// TIA Portal V17 export
// export: Created 2023-04-06T09:22:57.7461834Z, ExportSetting WithDefaults, DisplayName Totally Integrated Automation Portal, DisplayVersion V17 Update 4, DisplayName TIA Portal Openness, DisplayVersion V17 Update 4, DisplayName TIA Portal Version Control Interface, DisplayVersion V17, DisplayName STEP 7 Professional, DisplayVersion V17 Update 4, DisplayName STEP 7 Safety, DisplayVersion V17, DisplayName WinCC Professional, DisplayVersion V17 Update 4
FUNCTION "BMS 1 (S)" : Void   // FC25, LAD
TITLE = ModBus TCP for CATL Battery
{ S7_Optimized_Access := 'TRUE' }
VERSION : 0.1
// stored: AutoNumber false, IsIECCheckEnabled false, SetENOAutomatically false, UDAEnableTagReadback false
   VAR_TEMP
      xSpare : Bool;
      BBwAlm1 : Word;
      BBwWarn1 : Word;
      BR01wAlm1 : Word;
      BR01wAlm2 : Word;
      BR01wAlm3 : Word;
      BR01wWarn1 : Word;
      BR02wAlm1 : Word;
      BR02wAlm2 : Word;
      BR02wAlm3 : Word;
      BR02wWarn1 : Word;
      BR03wAlm1 : Word;
      BR03wAlm2 : Word;
      BR03wAlm3 : Word;
      BR03wWarn1 : Word;
      BR04wAlm1 : Word;
      BR04wAlm2 : Word;
      BR04wAlm3 : Word;
      BR04wWarn1 : Word;
      BR05wAlm1 : Word;
      BR05wAlm2 : Word;
      BR05wAlm3 : Word;
      BR05wWarn1 : Word;
      BR06wAlm1 : Word;
      BR06wAlm2 : Word;
      BR06wAlm3 : Word;
      BR06wWarn1 : Word;
      BR07wAlm1 : Word;
      BR07wAlm2 : Word;
      BR07wAlm3 : Word;
      BR07wWarn1 : Word;
      BR08wAlm1 : Word;
      BR08wAlm2 : Word;
      BR08wAlm3 : Word;
      BR08wWarn1 : Word;
      BR09wAlm1 : Word;
      BR09wAlm2 : Word;
      BR09wAlm3 : Word;
      BR09wWarn1 : Word;
      BR10wAlm1 : Word;
      BR10wAlm2 : Word;
      BR10wAlm3 : Word;
      BR10wWarn1 : Word;
      BR11wAlm1 : Word;
      BR11wAlm2 : Word;
      BR11wAlm3 : Word;
      BR11wWarn1 : Word;
      BR12wAlm1 : Word;
      BR12wAlm2 : Word;
      BR12wAlm3 : Word;
      BR12wWarn1 : Word;
   END_VAR
   VAR_TEMP   // added for the SCL form of the ladder/FBD networks
      _w1 : Bool;
   END_VAR
BEGIN

REGION Network 1: Function Modbus Client
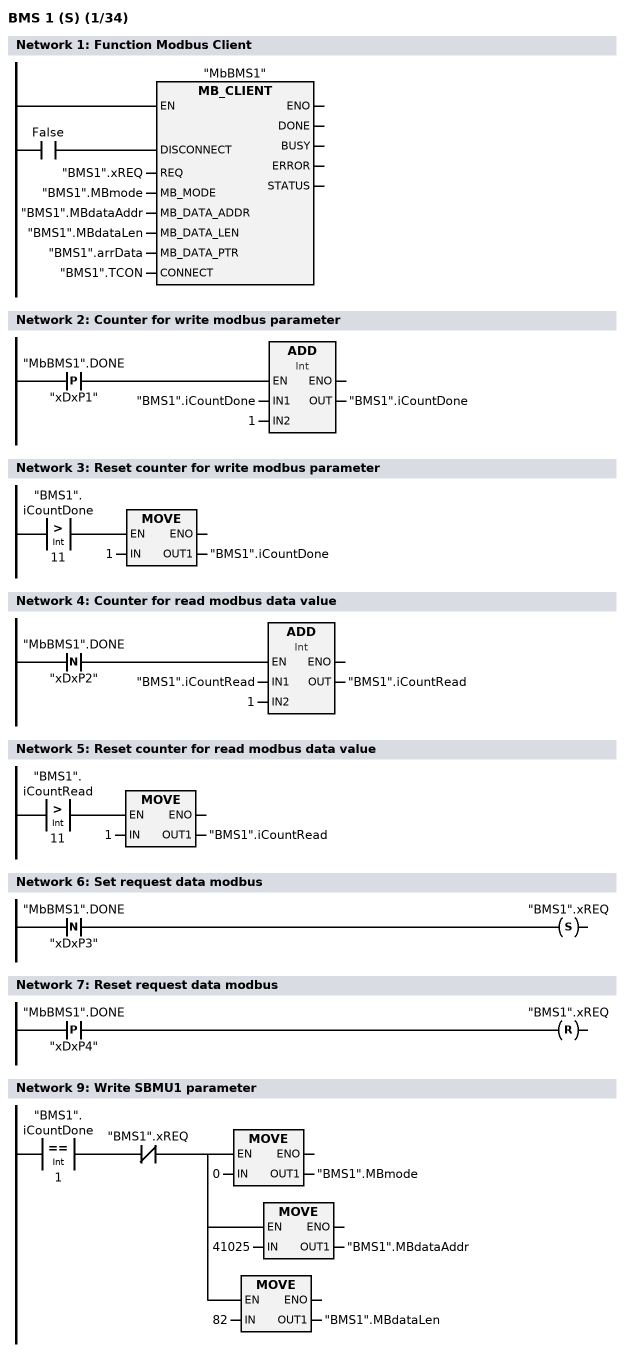
   RUNG wire#powerrail
      "MbBMS1".MB_CLIENT(DISCONNECT := wire#w1, REQ := "BMS1".xREQ, MB_MODE := "BMS1".MBmode, MB_DATA_ADDR := "BMS1".MBdataAddr, MB_DATA_LEN := "BMS1".MBdataLen, MB_DATA_PTR := "BMS1".arrData, CONNECT := "BMS1".TCON, DONE =>, BUSY =>, ERROR =>, STATUS =>)
   END_RUNG
   RUNG wire#powerrail
      Contact( False )
   END_RUNG wire#w1
   // the same network as SCL:
   "MbBMS1"(DISCONNECT := False,   // MB_CLIENT
            REQ := "BMS1".xREQ,
            MB_MODE := "BMS1".MBmode,
            MB_DATA_ADDR := "BMS1".MBdataAddr,
            MB_DATA_LEN := "BMS1".MBdataLen,
            MB_DATA_PTR := "BMS1".arrData,
            CONNECT := "BMS1".TCON);
END_REGION

REGION Network 2: Counter for write modbus parameter
   RUNG wire#powerrail
      P_Contact(operand := "MbBMS1".DONE, bit := "xDxP1")
      { S7_Templates := "SrcType := Int" } Add(in1 := "BMS1".iCountDone, in2 := 1, out => "BMS1".iCountDone)
   END_RUNG
   // the same network as SCL:
   #_w1 := "MbBMS1".DONE AND NOT "xDxP1";   // rising edge of "MbBMS1".DONE
   "xDxP1" := "MbBMS1".DONE;
   IF #_w1 THEN "BMS1".iCountDone := "BMS1".iCountDone + 1; END_IF;
END_REGION

REGION Network 3: Reset counter for write modbus parameter
   RUNG wire#powerrail
      { S7_Templates := "SrcType := Int" } GT_Contact(in1 := "BMS1".iCountDone, in2 := 11)
      Move(in := 1, out1 => "BMS1".iCountDone)
   END_RUNG
   // the same network as SCL:
   IF "BMS1".iCountDone > 11 THEN "BMS1".iCountDone := 1; END_IF;
END_REGION

REGION Network 4: Counter for read modbus data value
   RUNG wire#powerrail
      N_Contact(operand := "MbBMS1".DONE, bit := "xDxP2")
      { S7_Templates := "SrcType := Int" } Add(in1 := "BMS1".iCountRead, in2 := 1, out => "BMS1".iCountRead)
   END_RUNG
   // the same network as SCL:
   #_w1 := NOT "MbBMS1".DONE AND "xDxP2";   // falling edge of "MbBMS1".DONE
   "xDxP2" := "MbBMS1".DONE;
   IF #_w1 THEN "BMS1".iCountRead := "BMS1".iCountRead + 1; END_IF;
END_REGION

REGION Network 5: Reset counter for read modbus data value
   RUNG wire#powerrail
      { S7_Templates := "SrcType := Int" } GT_Contact(in1 := "BMS1".iCountRead, in2 := 11)
      Move(in := 1, out1 => "BMS1".iCountRead)
   END_RUNG
   // the same network as SCL:
   IF "BMS1".iCountRead > 11 THEN "BMS1".iCountRead := 1; END_IF;
END_REGION

REGION Network 6: Set request data modbus
   RUNG wire#powerrail
      N_Contact(operand := "MbBMS1".DONE, bit := "xDxP3")
      S_Coil( "BMS1".xREQ )
   END_RUNG
   // the same network as SCL:
   #_w1 := NOT "MbBMS1".DONE AND "xDxP3";   // falling edge of "MbBMS1".DONE
   "xDxP3" := "MbBMS1".DONE;
   IF #_w1 THEN "BMS1".xREQ := TRUE; END_IF;
END_REGION

REGION Network 7: Reset request data modbus
   RUNG wire#powerrail
      P_Contact(operand := "MbBMS1".DONE, bit := "xDxP4")
      R_Coil( "BMS1".xREQ )
   END_RUNG
   // the same network as SCL:
   #_w1 := "MbBMS1".DONE AND NOT "xDxP4";   // rising edge of "MbBMS1".DONE
   "xDxP4" := "MbBMS1".DONE;
   IF #_w1 THEN "BMS1".xREQ := FALSE; END_IF;
END_REGION

REGION Network 9: Write SBMU1 parameter
   RUNG wire#powerrail
      { S7_Templates := "SrcType := Int" } EQ_Contact(in1 := "BMS1".iCountDone, in2 := 1)
      I_Contact( "BMS1".xREQ )
      wire#w1
      Move(in := 0, out1 => "BMS1".MBmode)
   END_RUNG
   RUNG wire#w1
      Move(in := 41025, out1 => "BMS1".MBdataAddr)
   END_RUNG
   RUNG wire#w1
      Move(in := 82, out1 => "BMS1".MBdataLen)
   END_RUNG
   // the same network as SCL:
   IF ("BMS1".iCountDone = 1) AND NOT "BMS1".xREQ THEN
       "BMS1".MBmode := 0;
       "BMS1".MBdataAddr := 41025;
       "BMS1".MBdataLen := 82;
   END_IF;
END_REGION

REGION Network 10: Read SBMU1 data value
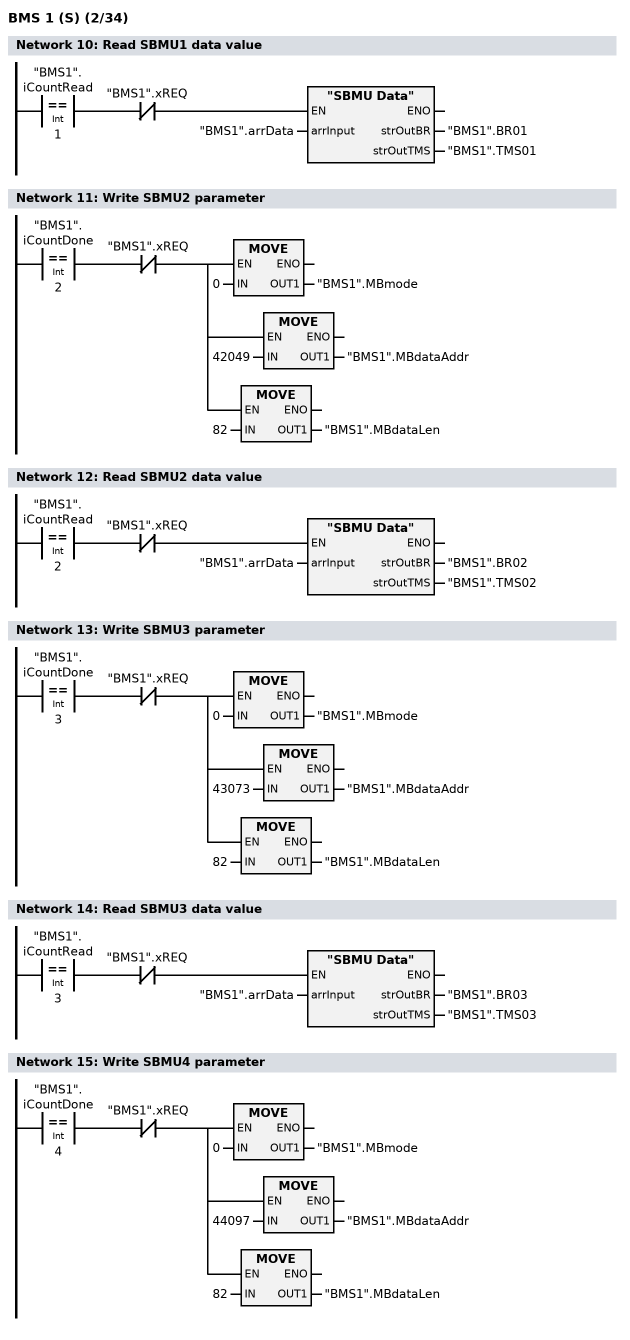
   RUNG wire#powerrail
      { S7_Templates := "SrcType := Int" } EQ_Contact(in1 := "BMS1".iCountRead, in2 := 1)
      I_Contact( "BMS1".xREQ )
      "SBMU Data"(arrInput := "BMS1".arrData, strOutBR => "BMS1".BR01, strOutTMS => "BMS1".TMS01)
   END_RUNG
   // the same network as SCL:
   IF ("BMS1".iCountRead = 1) AND NOT "BMS1".xREQ THEN
       "SBMU Data"(arrInput := "BMS1".arrData, strOutBR => "BMS1".BR01, strOutTMS => "BMS1".TMS01);
   END_IF;
END_REGION

REGION Network 11: Write SBMU2 parameter
   RUNG wire#powerrail
      { S7_Templates := "SrcType := Int" } EQ_Contact(in1 := "BMS1".iCountDone, in2 := 2)
      I_Contact( "BMS1".xREQ )
      wire#w1
      Move(in := 0, out1 => "BMS1".MBmode)
   END_RUNG
   RUNG wire#w1
      Move(in := 42049, out1 => "BMS1".MBdataAddr)
   END_RUNG
   RUNG wire#w1
      Move(in := 82, out1 => "BMS1".MBdataLen)
   END_RUNG
   // the same network as SCL:
   IF ("BMS1".iCountDone = 2) AND NOT "BMS1".xREQ THEN
       "BMS1".MBmode := 0;
       "BMS1".MBdataAddr := 42049;
       "BMS1".MBdataLen := 82;
   END_IF;
END_REGION

REGION Network 12: Read SBMU2 data value
   RUNG wire#powerrail
      { S7_Templates := "SrcType := Int" } EQ_Contact(in1 := "BMS1".iCountRead, in2 := 2)
      I_Contact( "BMS1".xREQ )
      "SBMU Data"(arrInput := "BMS1".arrData, strOutBR => "BMS1".BR02, strOutTMS => "BMS1".TMS02)
   END_RUNG
   // the same network as SCL:
   IF ("BMS1".iCountRead = 2) AND NOT "BMS1".xREQ THEN
       "SBMU Data"(arrInput := "BMS1".arrData, strOutBR => "BMS1".BR02, strOutTMS => "BMS1".TMS02);
   END_IF;
END_REGION

REGION Network 13: Write SBMU3 parameter
   RUNG wire#powerrail
      { S7_Templates := "SrcType := Int" } EQ_Contact(in1 := "BMS1".iCountDone, in2 := 3)
      I_Contact( "BMS1".xREQ )
      wire#w1
      Move(in := 0, out1 => "BMS1".MBmode)
   END_RUNG
   RUNG wire#w1
      Move(in := 43073, out1 => "BMS1".MBdataAddr)
   END_RUNG
   RUNG wire#w1
      Move(in := 82, out1 => "BMS1".MBdataLen)
   END_RUNG
   // the same network as SCL:
   IF ("BMS1".iCountDone = 3) AND NOT "BMS1".xREQ THEN
       "BMS1".MBmode := 0;
       "BMS1".MBdataAddr := 43073;
       "BMS1".MBdataLen := 82;
   END_IF;
END_REGION

REGION Network 14: Read SBMU3 data value
   RUNG wire#powerrail
      { S7_Templates := "SrcType := Int" } EQ_Contact(in1 := "BMS1".iCountRead, in2 := 3)
      I_Contact( "BMS1".xREQ )
      "SBMU Data"(arrInput := "BMS1".arrData, strOutBR => "BMS1".BR03, strOutTMS => "BMS1".TMS03)
   END_RUNG
   // the same network as SCL:
   IF ("BMS1".iCountRead = 3) AND NOT "BMS1".xREQ THEN
       "SBMU Data"(arrInput := "BMS1".arrData, strOutBR => "BMS1".BR03, strOutTMS => "BMS1".TMS03);
   END_IF;
END_REGION

REGION Network 15: Write SBMU4 parameter
   RUNG wire#powerrail
      { S7_Templates := "SrcType := Int" } EQ_Contact(in1 := "BMS1".iCountDone, in2 := 4)
      I_Contact( "BMS1".xREQ )
      wire#w1
      Move(in := 0, out1 => "BMS1".MBmode)
   END_RUNG
   RUNG wire#w1
      Move(in := 44097, out1 => "BMS1".MBdataAddr)
   END_RUNG
   RUNG wire#w1
      Move(in := 82, out1 => "BMS1".MBdataLen)
   END_RUNG
   // the same network as SCL:
   IF ("BMS1".iCountDone = 4) AND NOT "BMS1".xREQ THEN
       "BMS1".MBmode := 0;
       "BMS1".MBdataAddr := 44097;
       "BMS1".MBdataLen := 82;
   END_IF;
END_REGION

REGION Network 16: Read SBMU4 data value
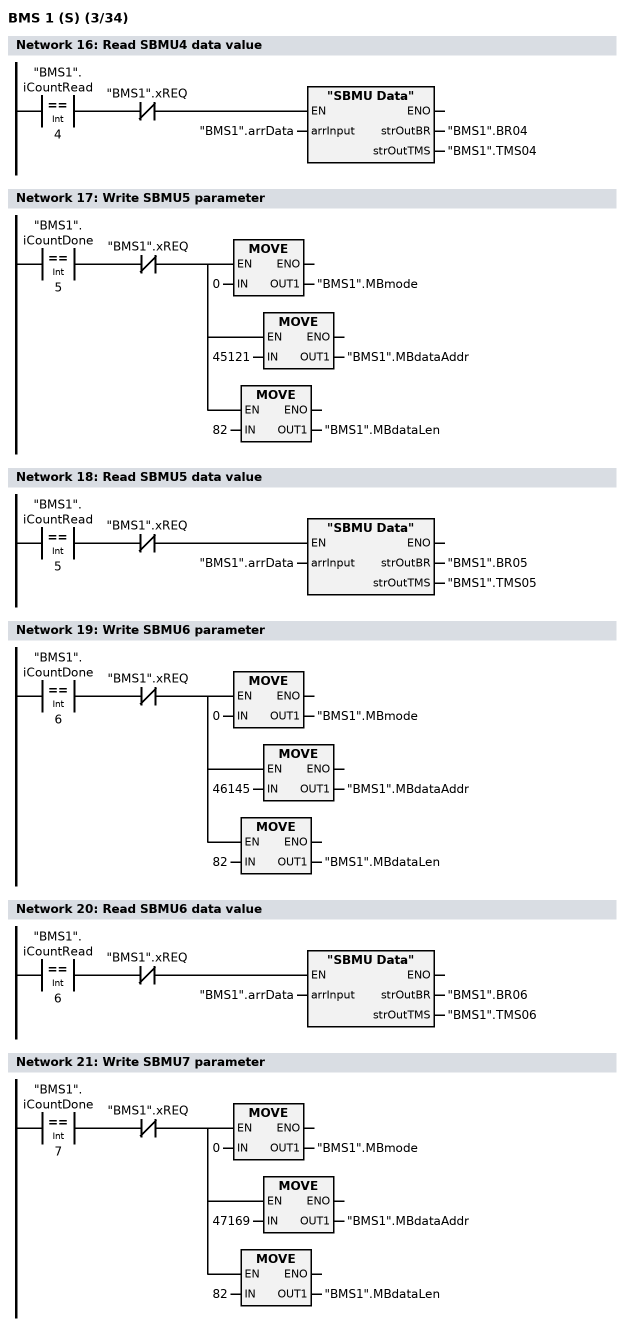
   RUNG wire#powerrail
      { S7_Templates := "SrcType := Int" } EQ_Contact(in1 := "BMS1".iCountRead, in2 := 4)
      I_Contact( "BMS1".xREQ )
      "SBMU Data"(arrInput := "BMS1".arrData, strOutBR => "BMS1".BR04, strOutTMS => "BMS1".TMS04)
   END_RUNG
   // the same network as SCL:
   IF ("BMS1".iCountRead = 4) AND NOT "BMS1".xREQ THEN
       "SBMU Data"(arrInput := "BMS1".arrData, strOutBR => "BMS1".BR04, strOutTMS => "BMS1".TMS04);
   END_IF;
END_REGION

REGION Network 17: Write SBMU5 parameter
   RUNG wire#powerrail
      { S7_Templates := "SrcType := Int" } EQ_Contact(in1 := "BMS1".iCountDone, in2 := 5)
      I_Contact( "BMS1".xREQ )
      wire#w1
      Move(in := 0, out1 => "BMS1".MBmode)
   END_RUNG
   RUNG wire#w1
      Move(in := 45121, out1 => "BMS1".MBdataAddr)
   END_RUNG
   RUNG wire#w1
      Move(in := 82, out1 => "BMS1".MBdataLen)
   END_RUNG
   // the same network as SCL:
   IF ("BMS1".iCountDone = 5) AND NOT "BMS1".xREQ THEN
       "BMS1".MBmode := 0;
       "BMS1".MBdataAddr := 45121;
       "BMS1".MBdataLen := 82;
   END_IF;
END_REGION

REGION Network 18: Read SBMU5 data value
   RUNG wire#powerrail
      { S7_Templates := "SrcType := Int" } EQ_Contact(in1 := "BMS1".iCountRead, in2 := 5)
      I_Contact( "BMS1".xREQ )
      "SBMU Data"(arrInput := "BMS1".arrData, strOutBR => "BMS1".BR05, strOutTMS => "BMS1".TMS05)
   END_RUNG
   // the same network as SCL:
   IF ("BMS1".iCountRead = 5) AND NOT "BMS1".xREQ THEN
       "SBMU Data"(arrInput := "BMS1".arrData, strOutBR => "BMS1".BR05, strOutTMS => "BMS1".TMS05);
   END_IF;
END_REGION

REGION Network 19: Write SBMU6 parameter
   RUNG wire#powerrail
      { S7_Templates := "SrcType := Int" } EQ_Contact(in1 := "BMS1".iCountDone, in2 := 6)
      I_Contact( "BMS1".xREQ )
      wire#w1
      Move(in := 0, out1 => "BMS1".MBmode)
   END_RUNG
   RUNG wire#w1
      Move(in := 46145, out1 => "BMS1".MBdataAddr)
   END_RUNG
   RUNG wire#w1
      Move(in := 82, out1 => "BMS1".MBdataLen)
   END_RUNG
   // the same network as SCL:
   IF ("BMS1".iCountDone = 6) AND NOT "BMS1".xREQ THEN
       "BMS1".MBmode := 0;
       "BMS1".MBdataAddr := 46145;
       "BMS1".MBdataLen := 82;
   END_IF;
END_REGION

REGION Network 20: Read SBMU6 data value
   RUNG wire#powerrail
      { S7_Templates := "SrcType := Int" } EQ_Contact(in1 := "BMS1".iCountRead, in2 := 6)
      I_Contact( "BMS1".xREQ )
      "SBMU Data"(arrInput := "BMS1".arrData, strOutBR => "BMS1".BR06, strOutTMS => "BMS1".TMS06)
   END_RUNG
   // the same network as SCL:
   IF ("BMS1".iCountRead = 6) AND NOT "BMS1".xREQ THEN
       "SBMU Data"(arrInput := "BMS1".arrData, strOutBR => "BMS1".BR06, strOutTMS => "BMS1".TMS06);
   END_IF;
END_REGION

REGION Network 21: Write SBMU7 parameter
   RUNG wire#powerrail
      { S7_Templates := "SrcType := Int" } EQ_Contact(in1 := "BMS1".iCountDone, in2 := 7)
      I_Contact( "BMS1".xREQ )
      wire#w1
      Move(in := 0, out1 => "BMS1".MBmode)
   END_RUNG
   RUNG wire#w1
      Move(in := 47169, out1 => "BMS1".MBdataAddr)
   END_RUNG
   RUNG wire#w1
      Move(in := 82, out1 => "BMS1".MBdataLen)
   END_RUNG
   // the same network as SCL:
   IF ("BMS1".iCountDone = 7) AND NOT "BMS1".xREQ THEN
       "BMS1".MBmode := 0;
       "BMS1".MBdataAddr := 47169;
       "BMS1".MBdataLen := 82;
   END_IF;
END_REGION

REGION Network 22: Read SBMU7 data value
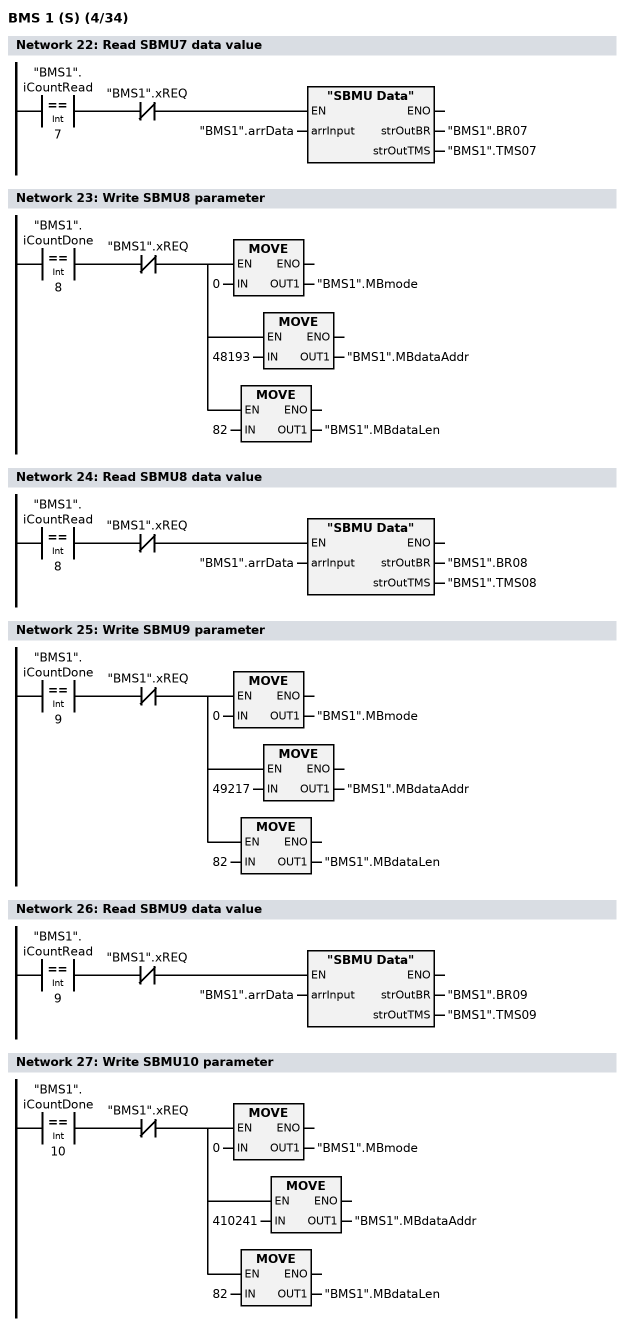
   RUNG wire#powerrail
      { S7_Templates := "SrcType := Int" } EQ_Contact(in1 := "BMS1".iCountRead, in2 := 7)
      I_Contact( "BMS1".xREQ )
      "SBMU Data"(arrInput := "BMS1".arrData, strOutBR => "BMS1".BR07, strOutTMS => "BMS1".TMS07)
   END_RUNG
   // the same network as SCL:
   IF ("BMS1".iCountRead = 7) AND NOT "BMS1".xREQ THEN
       "SBMU Data"(arrInput := "BMS1".arrData, strOutBR => "BMS1".BR07, strOutTMS => "BMS1".TMS07);
   END_IF;
END_REGION

REGION Network 23: Write SBMU8 parameter
   RUNG wire#powerrail
      { S7_Templates := "SrcType := Int" } EQ_Contact(in1 := "BMS1".iCountDone, in2 := 8)
      I_Contact( "BMS1".xREQ )
      wire#w1
      Move(in := 0, out1 => "BMS1".MBmode)
   END_RUNG
   RUNG wire#w1
      Move(in := 48193, out1 => "BMS1".MBdataAddr)
   END_RUNG
   RUNG wire#w1
      Move(in := 82, out1 => "BMS1".MBdataLen)
   END_RUNG
   // the same network as SCL:
   IF ("BMS1".iCountDone = 8) AND NOT "BMS1".xREQ THEN
       "BMS1".MBmode := 0;
       "BMS1".MBdataAddr := 48193;
       "BMS1".MBdataLen := 82;
   END_IF;
END_REGION

REGION Network 24: Read SBMU8 data value
   RUNG wire#powerrail
      { S7_Templates := "SrcType := Int" } EQ_Contact(in1 := "BMS1".iCountRead, in2 := 8)
      I_Contact( "BMS1".xREQ )
      "SBMU Data"(arrInput := "BMS1".arrData, strOutBR => "BMS1".BR08, strOutTMS => "BMS1".TMS08)
   END_RUNG
   // the same network as SCL:
   IF ("BMS1".iCountRead = 8) AND NOT "BMS1".xREQ THEN
       "SBMU Data"(arrInput := "BMS1".arrData, strOutBR => "BMS1".BR08, strOutTMS => "BMS1".TMS08);
   END_IF;
END_REGION

REGION Network 25: Write SBMU9 parameter
   RUNG wire#powerrail
      { S7_Templates := "SrcType := Int" } EQ_Contact(in1 := "BMS1".iCountDone, in2 := 9)
      I_Contact( "BMS1".xREQ )
      wire#w1
      Move(in := 0, out1 => "BMS1".MBmode)
   END_RUNG
   RUNG wire#w1
      Move(in := 49217, out1 => "BMS1".MBdataAddr)
   END_RUNG
   RUNG wire#w1
      Move(in := 82, out1 => "BMS1".MBdataLen)
   END_RUNG
   // the same network as SCL:
   IF ("BMS1".iCountDone = 9) AND NOT "BMS1".xREQ THEN
       "BMS1".MBmode := 0;
       "BMS1".MBdataAddr := 49217;
       "BMS1".MBdataLen := 82;
   END_IF;
END_REGION

REGION Network 26: Read SBMU9 data value
   RUNG wire#powerrail
      { S7_Templates := "SrcType := Int" } EQ_Contact(in1 := "BMS1".iCountRead, in2 := 9)
      I_Contact( "BMS1".xREQ )
      "SBMU Data"(arrInput := "BMS1".arrData, strOutBR => "BMS1".BR09, strOutTMS => "BMS1".TMS09)
   END_RUNG
   // the same network as SCL:
   IF ("BMS1".iCountRead = 9) AND NOT "BMS1".xREQ THEN
       "SBMU Data"(arrInput := "BMS1".arrData, strOutBR => "BMS1".BR09, strOutTMS => "BMS1".TMS09);
   END_IF;
END_REGION

REGION Network 27: Write SBMU10 parameter
   RUNG wire#powerrail
      { S7_Templates := "SrcType := Int" } EQ_Contact(in1 := "BMS1".iCountDone, in2 := 10)
      I_Contact( "BMS1".xREQ )
      wire#w1
      Move(in := 0, out1 => "BMS1".MBmode)
   END_RUNG
   RUNG wire#w1
      Move(in := 410241, out1 => "BMS1".MBdataAddr)
   END_RUNG
   RUNG wire#w1
      Move(in := 82, out1 => "BMS1".MBdataLen)
   END_RUNG
   // the same network as SCL:
   IF ("BMS1".iCountDone = 10) AND NOT "BMS1".xREQ THEN
       "BMS1".MBmode := 0;
       "BMS1".MBdataAddr := 410241;
       "BMS1".MBdataLen := 82;
   END_IF;
END_REGION

REGION Network 28: Read SBMU10 data value
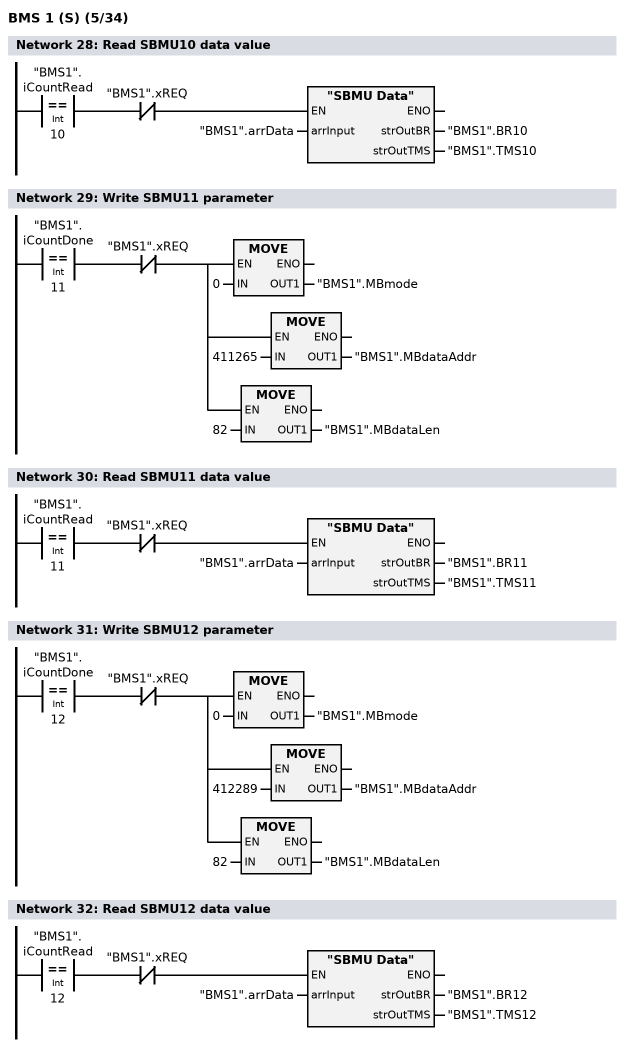
   RUNG wire#powerrail
      { S7_Templates := "SrcType := Int" } EQ_Contact(in1 := "BMS1".iCountRead, in2 := 10)
      I_Contact( "BMS1".xREQ )
      "SBMU Data"(arrInput := "BMS1".arrData, strOutBR => "BMS1".BR10, strOutTMS => "BMS1".TMS10)
   END_RUNG
   // the same network as SCL:
   IF ("BMS1".iCountRead = 10) AND NOT "BMS1".xREQ THEN
       "SBMU Data"(arrInput := "BMS1".arrData, strOutBR => "BMS1".BR10, strOutTMS => "BMS1".TMS10);
   END_IF;
END_REGION

REGION Network 29: Write SBMU11 parameter
   RUNG wire#powerrail
      { S7_Templates := "SrcType := Int" } EQ_Contact(in1 := "BMS1".iCountDone, in2 := 11)
      I_Contact( "BMS1".xREQ )
      wire#w1
      Move(in := 0, out1 => "BMS1".MBmode)
   END_RUNG
   RUNG wire#w1
      Move(in := 411265, out1 => "BMS1".MBdataAddr)
   END_RUNG
   RUNG wire#w1
      Move(in := 82, out1 => "BMS1".MBdataLen)
   END_RUNG
   // the same network as SCL:
   IF ("BMS1".iCountDone = 11) AND NOT "BMS1".xREQ THEN
       "BMS1".MBmode := 0;
       "BMS1".MBdataAddr := 411265;
       "BMS1".MBdataLen := 82;
   END_IF;
END_REGION

REGION Network 30: Read SBMU11 data value
   RUNG wire#powerrail
      { S7_Templates := "SrcType := Int" } EQ_Contact(in1 := "BMS1".iCountRead, in2 := 11)
      I_Contact( "BMS1".xREQ )
      "SBMU Data"(arrInput := "BMS1".arrData, strOutBR => "BMS1".BR11, strOutTMS => "BMS1".TMS11)
   END_RUNG
   // the same network as SCL:
   IF ("BMS1".iCountRead = 11) AND NOT "BMS1".xREQ THEN
       "SBMU Data"(arrInput := "BMS1".arrData, strOutBR => "BMS1".BR11, strOutTMS => "BMS1".TMS11);
   END_IF;
END_REGION

REGION Network 31: Write SBMU12 parameter
   RUNG wire#powerrail
      { S7_Templates := "SrcType := Int" } EQ_Contact(in1 := "BMS1".iCountDone, in2 := 12)
      I_Contact( "BMS1".xREQ )
      wire#w1
      Move(in := 0, out1 => "BMS1".MBmode)
   END_RUNG
   RUNG wire#w1
      Move(in := 412289, out1 => "BMS1".MBdataAddr)
   END_RUNG
   RUNG wire#w1
      Move(in := 82, out1 => "BMS1".MBdataLen)
   END_RUNG
   // the same network as SCL:
   IF ("BMS1".iCountDone = 12) AND NOT "BMS1".xREQ THEN
       "BMS1".MBmode := 0;
       "BMS1".MBdataAddr := 412289;
       "BMS1".MBdataLen := 82;
   END_IF;
END_REGION

REGION Network 32: Read SBMU12 data value
   RUNG wire#powerrail
      { S7_Templates := "SrcType := Int" } EQ_Contact(in1 := "BMS1".iCountRead, in2 := 12)
      I_Contact( "BMS1".xREQ )
      "SBMU Data"(arrInput := "BMS1".arrData, strOutBR => "BMS1".BR12, strOutTMS => "BMS1".TMS12)
   END_RUNG
   // the same network as SCL:
   IF ("BMS1".iCountRead = 12) AND NOT "BMS1".xREQ THEN
       "SBMU Data"(arrInput := "BMS1".arrData, strOutBR => "BMS1".BR12, strOutTMS => "BMS1".TMS12);
   END_IF;
END_REGION

REGION Network 34: Write Command from EMS
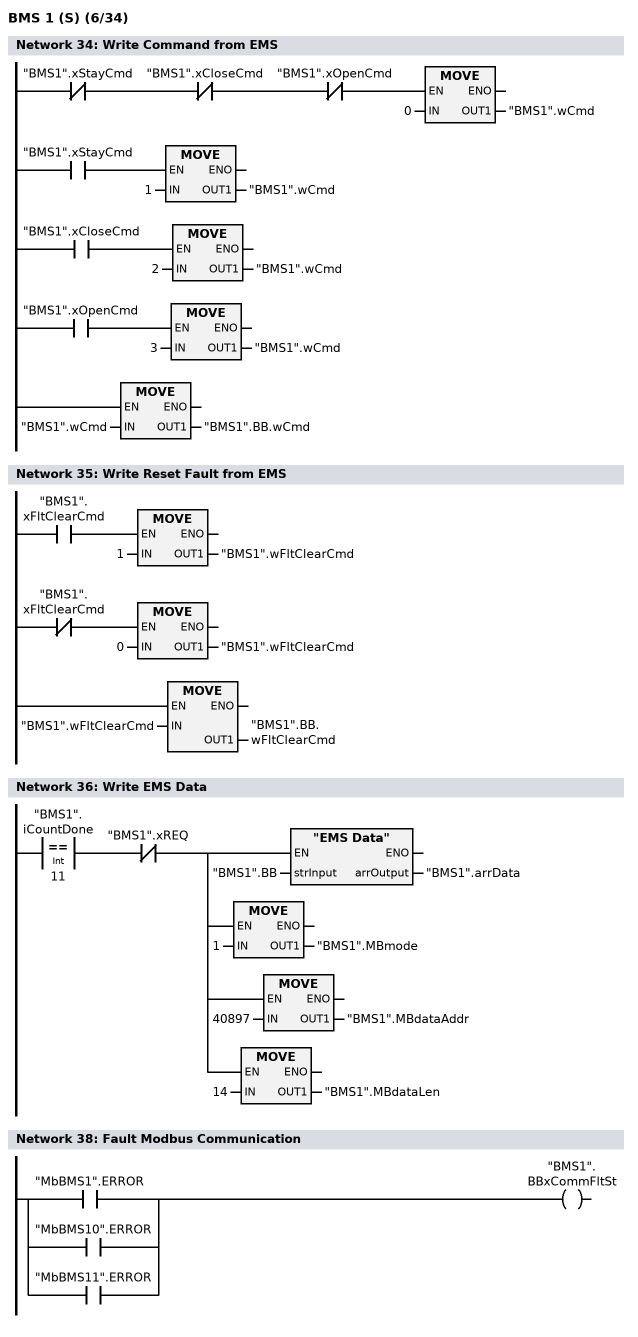
   RUNG wire#powerrail
      I_Contact( "BMS1".xStayCmd )
      I_Contact( "BMS1".xCloseCmd )
      I_Contact( "BMS1".xOpenCmd )
      Move(in := 0, out1 => "BMS1".wCmd)
   END_RUNG
   RUNG wire#powerrail
      Contact( "BMS1".xStayCmd )
      Move(in := 1, out1 => "BMS1".wCmd)
   END_RUNG
   RUNG wire#powerrail
      Contact( "BMS1".xCloseCmd )
      Move(in := 2, out1 => "BMS1".wCmd)
   END_RUNG
   RUNG wire#powerrail
      Contact( "BMS1".xOpenCmd )
      Move(in := 3, out1 => "BMS1".wCmd)
   END_RUNG
   RUNG wire#powerrail
      Move(in := "BMS1".wCmd, out1 => "BMS1".BB.wCmd)
   END_RUNG
   // the same network as SCL:
   IF NOT "BMS1".xStayCmd AND NOT "BMS1".xCloseCmd AND NOT "BMS1".xOpenCmd THEN "BMS1".wCmd := 0; END_IF;
   IF "BMS1".xStayCmd THEN "BMS1".wCmd := 1; END_IF;
   IF "BMS1".xCloseCmd THEN "BMS1".wCmd := 2; END_IF;
   IF "BMS1".xOpenCmd THEN "BMS1".wCmd := 3; END_IF;
   "BMS1".BB.wCmd := "BMS1".wCmd;
END_REGION

REGION Network 35: Write Reset Fault from EMS
   RUNG wire#powerrail
      Contact( "BMS1".xFltClearCmd )
      Move(in := 1, out1 => "BMS1".wFltClearCmd)
   END_RUNG
   RUNG wire#powerrail
      I_Contact( "BMS1".xFltClearCmd )
      Move(in := 0, out1 => "BMS1".wFltClearCmd)
   END_RUNG
   RUNG wire#powerrail
      Move(in := "BMS1".wFltClearCmd, out1 => "BMS1".BB.wFltClearCmd)
   END_RUNG
   // the same network as SCL:
   IF "BMS1".xFltClearCmd THEN "BMS1".wFltClearCmd := 1; END_IF;
   IF NOT "BMS1".xFltClearCmd THEN "BMS1".wFltClearCmd := 0; END_IF;
   "BMS1".BB.wFltClearCmd := "BMS1".wFltClearCmd;
END_REGION

REGION Network 36: Write EMS Data
   RUNG wire#powerrail
      { S7_Templates := "SrcType := Int" } EQ_Contact(in1 := "BMS1".iCountDone, in2 := 11)
      I_Contact( "BMS1".xREQ )
      wire#w1
      "EMS Data"(strInput := "BMS1".BB, arrOutput => "BMS1".arrData)
   END_RUNG
   RUNG wire#w1
      Move(in := 1, out1 => "BMS1".MBmode)
   END_RUNG
   RUNG wire#w1
      Move(in := 40897, out1 => "BMS1".MBdataAddr)
   END_RUNG
   RUNG wire#w1
      Move(in := 14, out1 => "BMS1".MBdataLen)
   END_RUNG
   // the same network as SCL:
   #_w1 := ("BMS1".iCountDone = 11) AND NOT "BMS1".xREQ;
   IF #_w1 THEN
       "EMS Data"(strInput := "BMS1".BB, arrOutput => "BMS1".arrData);
       "BMS1".MBmode := 1;
       "BMS1".MBdataAddr := 40897;
       "BMS1".MBdataLen := 14;
   END_IF;
END_REGION

REGION Network 38: Fault Modbus Communication
   RUNG wire#powerrail
      Contact( "MbBMS1".ERROR )
      wire#w1
      Coil( "BMS1".BBxCommFltSt )
   END_RUNG
   RUNG wire#powerrail
      Contact( "MbBMS10".ERROR )
   END_RUNG wire#w1
   RUNG wire#powerrail
      Contact( "MbBMS11".ERROR )
   END_RUNG wire#w1
   // the same network as SCL:
   "BMS1".BBxCommFltSt := "MbBMS1".ERROR OR "MbBMS10".ERROR OR "MbBMS11".ERROR;
END_REGION

REGION Network 40
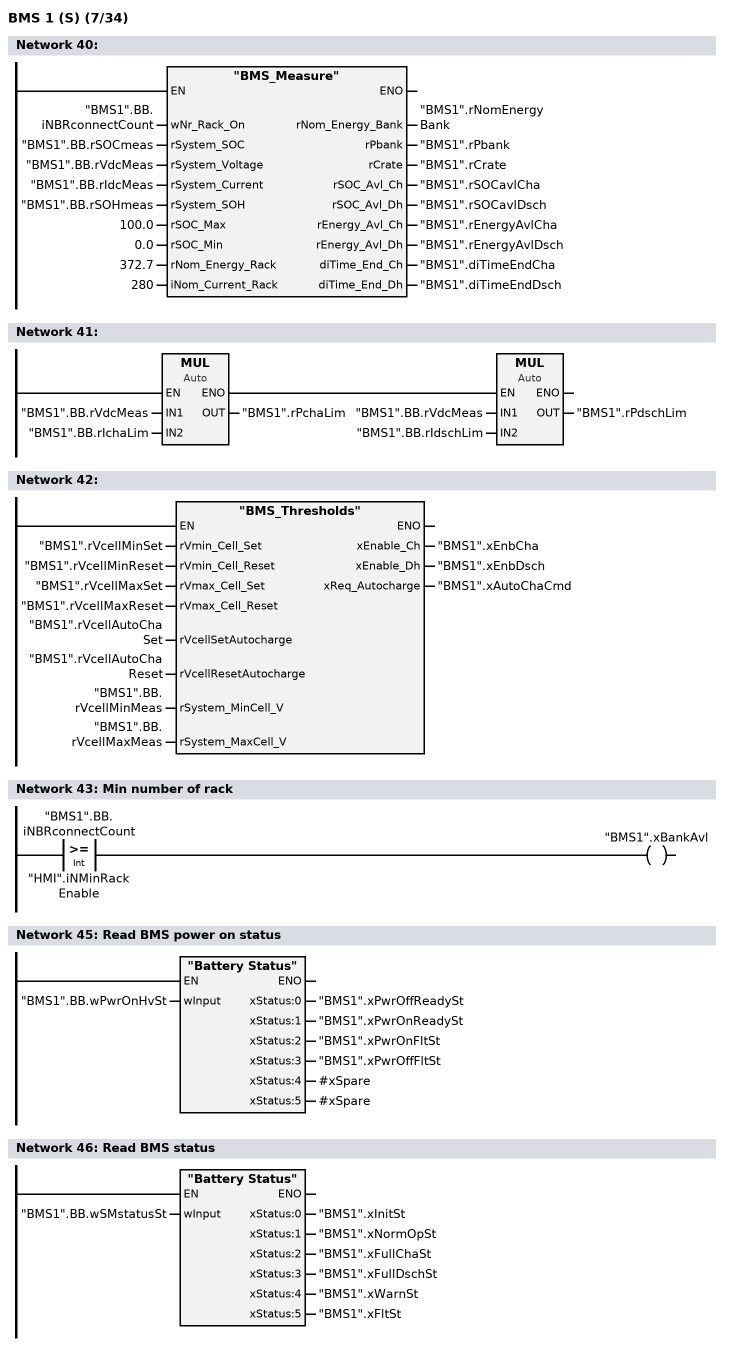
   RUNG wire#powerrail
      "BMS_Measure"(wNr_Rack_On := "BMS1".BB.iNBRconnectCount, rSystem_SOC := "BMS1".BB.rSOCmeas, rSystem_Voltage := "BMS1".BB.rVdcMeas, rSystem_Current := "BMS1".BB.rIdcMeas, rSystem_SOH := "BMS1".BB.rSOHmeas, rSOC_Max := 100.0, rSOC_Min := 0.0, rNom_Energy_Rack := 372.7, iNom_Current_Rack := 280, rNom_Energy_Bank => "BMS1".rNomEnergyBank, rPbank => "BMS1".rPbank, rCrate => "BMS1".rCrate, rSOC_Avl_Ch => "BMS1".rSOCavlCha, rSOC_Avl_Dh => "BMS1".rSOCavlDsch, rEnergy_Avl_Ch => "BMS1".rEnergyAvlCha, rEnergy_Avl_Dh => "BMS1".rEnergyAvlDsch, diTime_End_Ch => "BMS1".diTimeEndCha, diTime_End_Dh => "BMS1".diTimeEndDsch)
   END_RUNG
   // the same network as SCL:
   "BMS_Measure"(wNr_Rack_On := "BMS1".BB.iNBRconnectCount,
                 rSystem_SOC := "BMS1".BB.rSOCmeas,
                 rSystem_Voltage := "BMS1".BB.rVdcMeas,
                 rSystem_Current := "BMS1".BB.rIdcMeas,
                 rSystem_SOH := "BMS1".BB.rSOHmeas,
                 rSOC_Max := 100.0,
                 rSOC_Min := 0.0,
                 rNom_Energy_Rack := 372.7,
                 iNom_Current_Rack := 280,
                 rNom_Energy_Bank => "BMS1".rNomEnergyBank,
                 rPbank => "BMS1".rPbank,
                 rCrate => "BMS1".rCrate,
                 rSOC_Avl_Ch => "BMS1".rSOCavlCha,
                 rSOC_Avl_Dh => "BMS1".rSOCavlDsch,
                 rEnergy_Avl_Ch => "BMS1".rEnergyAvlCha,
                 rEnergy_Avl_Dh => "BMS1".rEnergyAvlDsch,
                 diTime_End_Ch => "BMS1".diTimeEndCha,
                 diTime_End_Dh => "BMS1".diTimeEndDsch);
END_REGION

REGION Network 41
   RUNG wire#powerrail
      Mul(in1 := "BMS1".BB.rVdcMeas, in2 := "BMS1".BB.rIchaLim, out => "BMS1".rPchaLim)
      Mul(in1 := "BMS1".BB.rVdcMeas, in2 := "BMS1".BB.rIdschLim, out => "BMS1".rPdschLim)
   END_RUNG
   // the same network as SCL:
   "BMS1".rPchaLim := "BMS1".BB.rVdcMeas * "BMS1".BB.rIchaLim;
   "BMS1".rPdschLim := "BMS1".BB.rVdcMeas * "BMS1".BB.rIdschLim;
END_REGION

REGION Network 42
   RUNG wire#powerrail
      "BMS_Thresholds"(rVmin_Cell_Set := "BMS1".rVcellMinSet, rVmin_Cell_Reset := "BMS1".rVcellMinReset, rVmax_Cell_Set := "BMS1".rVcellMaxSet, rVmax_Cell_Reset := "BMS1".rVcellMaxReset, rVcellSetAutocharge := "BMS1".rVcellAutoChaSet, rVcellResetAutocharge := "BMS1".rVcellAutoChaReset, rSystem_MinCell_V := "BMS1".BB.rVcellMinMeas, rSystem_MaxCell_V := "BMS1".BB.rVcellMaxMeas, xEnable_Ch => "BMS1".xEnbCha, xEnable_Dh => "BMS1".xEnbDsch, xReq_Autocharge => "BMS1".xAutoChaCmd)
   END_RUNG
   // the same network as SCL:
   "BMS_Thresholds"(rVmin_Cell_Set := "BMS1".rVcellMinSet,
                    rVmin_Cell_Reset := "BMS1".rVcellMinReset,
                    rVmax_Cell_Set := "BMS1".rVcellMaxSet,
                    rVmax_Cell_Reset := "BMS1".rVcellMaxReset,
                    rVcellSetAutocharge := "BMS1".rVcellAutoChaSet,
                    rVcellResetAutocharge := "BMS1".rVcellAutoChaReset,
                    rSystem_MinCell_V := "BMS1".BB.rVcellMinMeas,
                    rSystem_MaxCell_V := "BMS1".BB.rVcellMaxMeas,
                    xEnable_Ch => "BMS1".xEnbCha,
                    xEnable_Dh => "BMS1".xEnbDsch,
                    xReq_Autocharge => "BMS1".xAutoChaCmd);
END_REGION

REGION Network 43: Min number of rack
   RUNG wire#powerrail
      { S7_Templates := "SrcType := Int" } GE_Contact(in1 := "BMS1".BB.iNBRconnectCount, in2 := "HMI".iNMinRackEnable)
      Coil( "BMS1".xBankAvl )
   END_RUNG
   // the same network as SCL:
   "BMS1".xBankAvl := "BMS1".BB.iNBRconnectCount >= "HMI".iNMinRackEnable;
END_REGION

REGION Network 45: Read BMS power on status
   RUNG wire#powerrail
      "Battery Status"(wInput := "BMS1".BB.wPwrOnHvSt, "xStatus:0" => "BMS1".xPwrOffReadySt, "xStatus:1" => "BMS1".xPwrOnReadySt, "xStatus:2" => "BMS1".xPwrOnFltSt, "xStatus:3" => "BMS1".xPwrOffFltSt, "xStatus:4" => #xSpare, "xStatus:5" => #xSpare)
   END_RUNG
   // the same network as SCL:
   "Battery Status"(wInput := "BMS1".BB.wPwrOnHvSt,
                    "xStatus:0" => "BMS1".xPwrOffReadySt,
                    "xStatus:1" => "BMS1".xPwrOnReadySt,
                    "xStatus:2" => "BMS1".xPwrOnFltSt,
                    "xStatus:3" => "BMS1".xPwrOffFltSt,
                    "xStatus:4" => #xSpare,
                    "xStatus:5" => #xSpare);
END_REGION

REGION Network 46: Read BMS status
   RUNG wire#powerrail
      "Battery Status"(wInput := "BMS1".BB.wSMstatusSt, "xStatus:0" => "BMS1".xInitSt, "xStatus:1" => "BMS1".xNormOpSt, "xStatus:2" => "BMS1".xFullChaSt, "xStatus:3" => "BMS1".xFullDschSt, "xStatus:4" => "BMS1".xWarnSt, "xStatus:5" => "BMS1".xFltSt)
   END_RUNG
   // the same network as SCL:
   "Battery Status"(wInput := "BMS1".BB.wSMstatusSt,
                    "xStatus:0" => "BMS1".xInitSt,
                    "xStatus:1" => "BMS1".xNormOpSt,
                    "xStatus:2" => "BMS1".xFullChaSt,
                    "xStatus:3" => "BMS1".xFullDschSt,
                    "xStatus:4" => "BMS1".xWarnSt,
                    "xStatus:5" => "BMS1".xFltSt);
END_REGION

REGION Network 48 (SCL): Rack Fault Status
   "BMS1".wRackFlt.%X0 := "BMS1".BR01xFltSt;
   "BMS1".wRackFlt.%X1 := "BMS1".BR02xFltSt;
   "BMS1".wRackFlt.%X2 := "BMS1".BR03xFltSt;
   "BMS1".wRackFlt.%X3 := "BMS1".BR04xFltSt;
   "BMS1".wRackFlt.%X4 := "BMS1".BR05xFltSt;
   "BMS1".wRackFlt.%X5 := "BMS1".BR06xFltSt;
   "BMS1".wRackFlt.%X6 := "BMS1".BR07xFltSt;
   "BMS1".wRackFlt.%X7 := "BMS1".BR08xFltSt;
   "BMS1".wRackFlt.%X8 := "BMS1".BR09xFltSt;
   "BMS1".wRackFlt.%X9 := "BMS1".BR10xFltSt;
END_REGION

REGION Network 49 (SCL): Rack On Status
   "BMS1".wRackOn.%X0 := "BMS1".BR01.xKposSt;
   "BMS1".wRackOn.%X1 := "BMS1".BR02.xKposSt;
   "BMS1".wRackOn.%X2 := "BMS1".BR03.xKposSt;
   "BMS1".wRackOn.%X3 := "BMS1".BR04.xKposSt;
   "BMS1".wRackOn.%X4 := "BMS1".BR05.xKposSt;
   "BMS1".wRackOn.%X5 := "BMS1".BR06.xKposSt;
   "BMS1".wRackOn.%X6 := "BMS1".BR07.xKposSt;
   "BMS1".wRackOn.%X7 := "BMS1".BR08.xKposSt;
   "BMS1".wRackOn.%X8 := "BMS1".BR09.xKposSt;
   "BMS1".wRackOn.%X9 := "BMS1".BR10.xKposSt;
END_REGION

REGION Network 50 (SCL): Status Switch Gear
   IF
       NOT "BMS1".BR01wAlm2.%X12 OR
       NOT "BMS1".BR02wAlm2.%X12 OR
       NOT "BMS1".BR03wAlm2.%X12 OR
       NOT "BMS1".BR04wAlm2.%X12 OR
       NOT "BMS1".BR05wAlm2.%X12 OR
       NOT "BMS1".BR06wAlm2.%X12 OR
       NOT "BMS1".BR07wAlm2.%X12 OR
       NOT "BMS1".BR08wAlm2.%X12 OR
       NOT "BMS1".BR09wAlm2.%X12 OR
       NOT "BMS1".BR10wAlm2.%X12 THEN

       "BMS1".xSwitchGearSt := True;
   ELSE
       "BMS1".xSwitchGearSt := False;
   END_IF;
END_REGION

REGION Network 52: Alarm MBMU
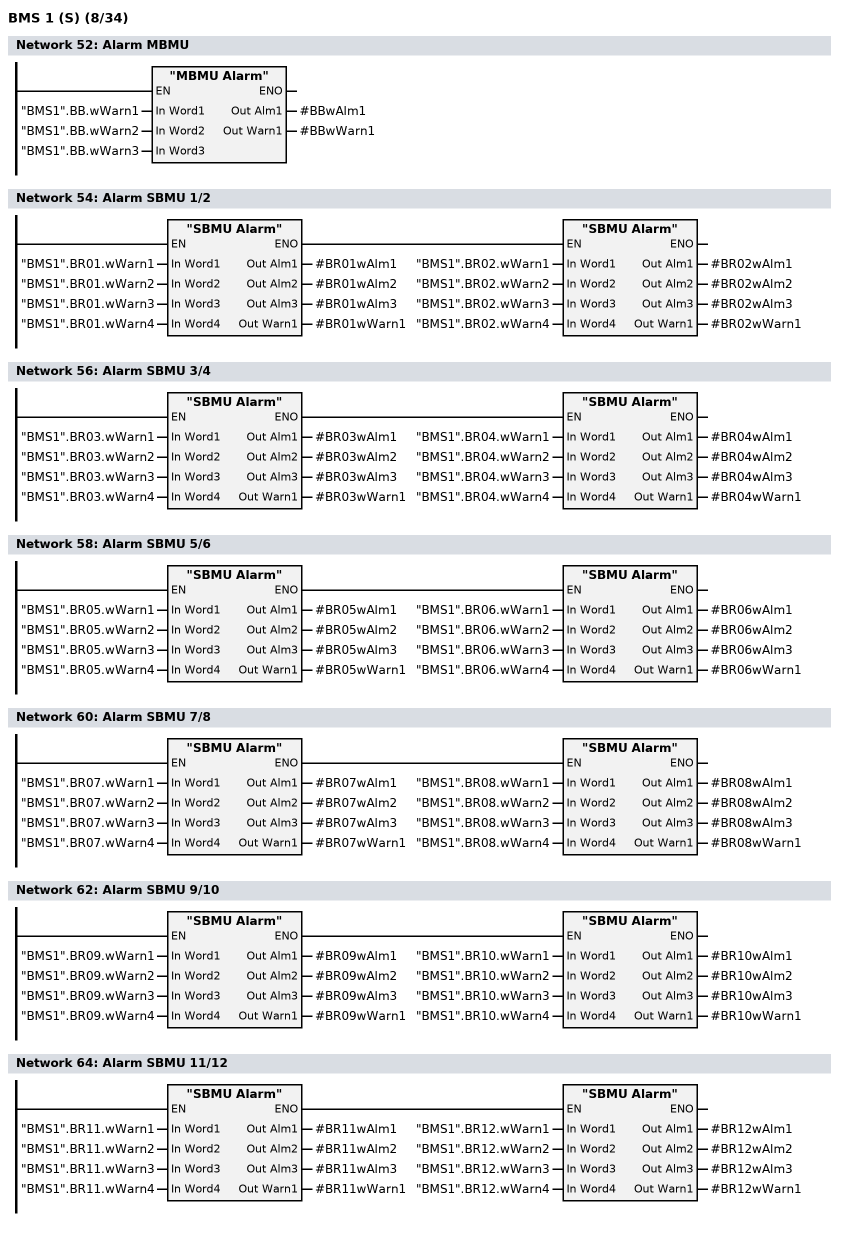
   RUNG wire#powerrail
      "MBMU Alarm"("In Word1" := "BMS1".BB.wWarn1, "In Word2" := "BMS1".BB.wWarn2, "In Word3" := "BMS1".BB.wWarn3, "Out Alm1" => #BBwAlm1, "Out Warn1" => #BBwWarn1)
   END_RUNG
   // the same network as SCL:
   "MBMU Alarm"("In Word1" := "BMS1".BB.wWarn1,
                "In Word2" := "BMS1".BB.wWarn2,
                "In Word3" := "BMS1".BB.wWarn3,
                "Out Alm1" => #BBwAlm1,
                "Out Warn1" => #BBwWarn1);
END_REGION

REGION Network 53 (SCL): Alarm MBMU to HMI
   IF "HMI".xBB1AlmDisable OR"HMI".xPEMSAlmDisable OR"HMI".xPIAlmDisable
   THEN
       "BMS1".BBwAlm1 := 0;
       "BMS1".BBwWarn1 := 0;
   ELSE
       "BMS1".BBwAlm1 := #BBwAlm1;
       "BMS1".BBwWarn1 := #BBwWarn1;
   END_IF;
END_REGION

REGION Network 54: Alarm SBMU 1/2
   RUNG wire#powerrail
      "SBMU Alarm"("In Word1" := "BMS1".BR01.wWarn1, "In Word2" := "BMS1".BR01.wWarn2, "In Word3" := "BMS1".BR01.wWarn3, "In Word4" := "BMS1".BR01.wWarn4, "Out Alm1" => #BR01wAlm1, "Out Alm2" => #BR01wAlm2, "Out Alm3" => #BR01wAlm3, "Out Warn1" => #BR01wWarn1)
      "SBMU Alarm"("In Word1" := "BMS1".BR02.wWarn1, "In Word2" := "BMS1".BR02.wWarn2, "In Word3" := "BMS1".BR02.wWarn3, "In Word4" := "BMS1".BR02.wWarn4, "Out Alm1" => #BR02wAlm1, "Out Alm2" => #BR02wAlm2, "Out Alm3" => #BR02wAlm3, "Out Warn1" => #BR02wWarn1)
   END_RUNG
   // the same network as SCL:
   "SBMU Alarm"("In Word1" := "BMS1".BR01.wWarn1,
                "In Word2" := "BMS1".BR01.wWarn2,
                "In Word3" := "BMS1".BR01.wWarn3,
                "In Word4" := "BMS1".BR01.wWarn4,
                "Out Alm1" => #BR01wAlm1,
                "Out Alm2" => #BR01wAlm2,
                "Out Alm3" => #BR01wAlm3,
                "Out Warn1" => #BR01wWarn1,
                ENO => #_w1);
   IF #_w1 THEN
       "SBMU Alarm"("In Word1" := "BMS1".BR02.wWarn1,
                    "In Word2" := "BMS1".BR02.wWarn2,
                    "In Word3" := "BMS1".BR02.wWarn3,
                    "In Word4" := "BMS1".BR02.wWarn4,
                    "Out Alm1" => #BR02wAlm1,
                    "Out Alm2" => #BR02wAlm2,
                    "Out Alm3" => #BR02wAlm3,
                    "Out Warn1" => #BR02wWarn1);
   END_IF;
END_REGION

REGION Network 55 (SCL): Alarm SBMU 1/2 to HMI
   IF "HMI".xBB1BR1AlmDisable OR "HMI".xBB1AlmDisable OR "HMI".xPEMSAlmDisable OR "HMI".xPIAlmDisable
   THEN
       "BMS1".BR01wAlm1 := 0;
       "BMS1".BR01wAlm2 := 0;
       "BMS1".BR01wAlm3 := 0;
       "BMS1".BR01wWarn1 := 0;
   ELSE
       "BMS1".BR01wAlm1 := #BR01wAlm1;
       "BMS1".BR01wAlm2 := #BR01wAlm2;
       "BMS1".BR01wAlm3 := #BR01wAlm3;
       "BMS1".BR01wWarn1 := #BR01wWarn1;
   END_IF;

   IF "HMI".xBB1BR2AlmDisable OR "HMI".xBB1AlmDisable OR "HMI".xPEMSAlmDisable OR "HMI".xPIAlmDisable
   THEN
       "BMS1".BR02wAlm1 := 0;
       "BMS1".BR02wAlm2 := 0;
       "BMS1".BR02wAlm3 := 0;
       "BMS1".BR02wWarn1 := 0;
   ELSE
       "BMS1".BR02wAlm1 := #BR02wAlm1;
       "BMS1".BR02wAlm2 := #BR02wAlm2;
       "BMS1".BR02wAlm3 := #BR02wAlm3;
       "BMS1".BR02wWarn1 := #BR02wWarn1;
   END_IF;
END_REGION

REGION Network 56: Alarm SBMU 3/4
   RUNG wire#powerrail
      "SBMU Alarm"("In Word1" := "BMS1".BR03.wWarn1, "In Word2" := "BMS1".BR03.wWarn2, "In Word3" := "BMS1".BR03.wWarn3, "In Word4" := "BMS1".BR03.wWarn4, "Out Alm1" => #BR03wAlm1, "Out Alm2" => #BR03wAlm2, "Out Alm3" => #BR03wAlm3, "Out Warn1" => #BR03wWarn1)
      "SBMU Alarm"("In Word1" := "BMS1".BR04.wWarn1, "In Word2" := "BMS1".BR04.wWarn2, "In Word3" := "BMS1".BR04.wWarn3, "In Word4" := "BMS1".BR04.wWarn4, "Out Alm1" => #BR04wAlm1, "Out Alm2" => #BR04wAlm2, "Out Alm3" => #BR04wAlm3, "Out Warn1" => #BR04wWarn1)
   END_RUNG
   // the same network as SCL:
   "SBMU Alarm"("In Word1" := "BMS1".BR03.wWarn1,
                "In Word2" := "BMS1".BR03.wWarn2,
                "In Word3" := "BMS1".BR03.wWarn3,
                "In Word4" := "BMS1".BR03.wWarn4,
                "Out Alm1" => #BR03wAlm1,
                "Out Alm2" => #BR03wAlm2,
                "Out Alm3" => #BR03wAlm3,
                "Out Warn1" => #BR03wWarn1,
                ENO => #_w1);
   IF #_w1 THEN
       "SBMU Alarm"("In Word1" := "BMS1".BR04.wWarn1,
                    "In Word2" := "BMS1".BR04.wWarn2,
                    "In Word3" := "BMS1".BR04.wWarn3,
                    "In Word4" := "BMS1".BR04.wWarn4,
                    "Out Alm1" => #BR04wAlm1,
                    "Out Alm2" => #BR04wAlm2,
                    "Out Alm3" => #BR04wAlm3,
                    "Out Warn1" => #BR04wWarn1);
   END_IF;
END_REGION

REGION Network 57 (SCL): Alarm SBMU 3/4 to HMI
   IF "HMI".xBB1BR3AlmDisable OR "HMI".xBB1AlmDisable OR "HMI".xPEMSAlmDisable OR "HMI".xPIAlmDisable
   THEN
       "BMS1".BR03wAlm1 := 0;
       "BMS1".BR03wAlm2 := 0;
       "BMS1".BR03wAlm3 := 0;
       "BMS1".BR03wWarn1 := 0;
   ELSE
       "BMS1".BR03wAlm1 := #BR03wAlm1;
       "BMS1".BR03wAlm2 := #BR03wAlm2;
       "BMS1".BR03wAlm3 := #BR03wAlm3;
       "BMS1".BR03wWarn1 := #BR03wWarn1;
   END_IF;

   IF "HMI".xBB1BR4AlmDisable OR "HMI".xBB1AlmDisable OR "HMI".xPEMSAlmDisable OR "HMI".xPIAlmDisable
   THEN
       "BMS1".BR04wAlm1 := 0;
       "BMS1".BR04wAlm2 := 0;
       "BMS1".BR04wAlm3 := 0;
       "BMS1".BR04wWarn1 := 0;
   ELSE
       "BMS1".BR04wAlm1 := #BR04wAlm1;
       "BMS1".BR04wAlm2 := #BR04wAlm2;
       "BMS1".BR04wAlm3 := #BR04wAlm3;
       "BMS1".BR04wWarn1 := #BR04wWarn1;
   END_IF;
END_REGION

REGION Network 58: Alarm SBMU 5/6
   RUNG wire#powerrail
      "SBMU Alarm"("In Word1" := "BMS1".BR05.wWarn1, "In Word2" := "BMS1".BR05.wWarn2, "In Word3" := "BMS1".BR05.wWarn3, "In Word4" := "BMS1".BR05.wWarn4, "Out Alm1" => #BR05wAlm1, "Out Alm2" => #BR05wAlm2, "Out Alm3" => #BR05wAlm3, "Out Warn1" => #BR05wWarn1)
      "SBMU Alarm"("In Word1" := "BMS1".BR06.wWarn1, "In Word2" := "BMS1".BR06.wWarn2, "In Word3" := "BMS1".BR06.wWarn3, "In Word4" := "BMS1".BR06.wWarn4, "Out Alm1" => #BR06wAlm1, "Out Alm2" => #BR06wAlm2, "Out Alm3" => #BR06wAlm3, "Out Warn1" => #BR06wWarn1)
   END_RUNG
   // the same network as SCL:
   "SBMU Alarm"("In Word1" := "BMS1".BR05.wWarn1,
                "In Word2" := "BMS1".BR05.wWarn2,
                "In Word3" := "BMS1".BR05.wWarn3,
                "In Word4" := "BMS1".BR05.wWarn4,
                "Out Alm1" => #BR05wAlm1,
                "Out Alm2" => #BR05wAlm2,
                "Out Alm3" => #BR05wAlm3,
                "Out Warn1" => #BR05wWarn1,
                ENO => #_w1);
   IF #_w1 THEN
       "SBMU Alarm"("In Word1" := "BMS1".BR06.wWarn1,
                    "In Word2" := "BMS1".BR06.wWarn2,
                    "In Word3" := "BMS1".BR06.wWarn3,
                    "In Word4" := "BMS1".BR06.wWarn4,
                    "Out Alm1" => #BR06wAlm1,
                    "Out Alm2" => #BR06wAlm2,
                    "Out Alm3" => #BR06wAlm3,
                    "Out Warn1" => #BR06wWarn1);
   END_IF;
END_REGION

REGION Network 59 (SCL): Alarm SBMU 5/6 to HMI
   IF "HMI".xBB1BR5AlmDisable OR "HMI".xBB1AlmDisable OR "HMI".xPEMSAlmDisable OR "HMI".xPIAlmDisable
   THEN
       "BMS1".BR05wAlm1 := 0;
       "BMS1".BR05wAlm2 := 0;
       "BMS1".BR05wAlm3 := 0;
       "BMS1".BR05wWarn1 := 0;
   ELSE
       "BMS1".BR05wAlm1 := #BR05wAlm1;
       "BMS1".BR05wAlm2 := #BR05wAlm2;
       "BMS1".BR05wAlm3 := #BR05wAlm3;
       "BMS1".BR05wWarn1 := #BR05wWarn1;
   END_IF;

   IF "HMI".xBB1BR6AlmDisable OR "HMI".xBB1AlmDisable OR "HMI".xPEMSAlmDisable OR "HMI".xPIAlmDisable
   THEN
       "BMS1".BR06wAlm1 := 0;
       "BMS1".BR06wAlm2 := 0;
       "BMS1".BR06wAlm3 := 0;
       "BMS1".BR06wWarn1 := 0;
   ELSE
       "BMS1".BR06wAlm1 := #BR06wAlm1;
       "BMS1".BR06wAlm2 := #BR06wAlm2;
       "BMS1".BR06wAlm3 := #BR06wAlm3;
       "BMS1".BR06wWarn1 := #BR06wWarn1;
   END_IF;
END_REGION

REGION Network 60: Alarm SBMU 7/8
   RUNG wire#powerrail
      "SBMU Alarm"("In Word1" := "BMS1".BR07.wWarn1, "In Word2" := "BMS1".BR07.wWarn2, "In Word3" := "BMS1".BR07.wWarn3, "In Word4" := "BMS1".BR07.wWarn4, "Out Alm1" => #BR07wAlm1, "Out Alm2" => #BR07wAlm2, "Out Alm3" => #BR07wAlm3, "Out Warn1" => #BR07wWarn1)
      "SBMU Alarm"("In Word1" := "BMS1".BR08.wWarn1, "In Word2" := "BMS1".BR08.wWarn2, "In Word3" := "BMS1".BR08.wWarn3, "In Word4" := "BMS1".BR08.wWarn4, "Out Alm1" => #BR08wAlm1, "Out Alm2" => #BR08wAlm2, "Out Alm3" => #BR08wAlm3, "Out Warn1" => #BR08wWarn1)
   END_RUNG
   // the same network as SCL:
   "SBMU Alarm"("In Word1" := "BMS1".BR07.wWarn1,
                "In Word2" := "BMS1".BR07.wWarn2,
                "In Word3" := "BMS1".BR07.wWarn3,
                "In Word4" := "BMS1".BR07.wWarn4,
                "Out Alm1" => #BR07wAlm1,
                "Out Alm2" => #BR07wAlm2,
                "Out Alm3" => #BR07wAlm3,
                "Out Warn1" => #BR07wWarn1,
                ENO => #_w1);
   IF #_w1 THEN
       "SBMU Alarm"("In Word1" := "BMS1".BR08.wWarn1,
                    "In Word2" := "BMS1".BR08.wWarn2,
                    "In Word3" := "BMS1".BR08.wWarn3,
                    "In Word4" := "BMS1".BR08.wWarn4,
                    "Out Alm1" => #BR08wAlm1,
                    "Out Alm2" => #BR08wAlm2,
                    "Out Alm3" => #BR08wAlm3,
                    "Out Warn1" => #BR08wWarn1);
   END_IF;
END_REGION

REGION Network 61 (SCL): Alarm SBMU 7/8 to HMI
   IF "HMI".xBB1BR7AlmDisable OR "HMI".xBB1AlmDisable OR "HMI".xPEMSAlmDisable OR "HMI".xPIAlmDisable
   THEN
       "BMS1".BR07wAlm1 := 0;
       "BMS1".BR07wAlm2 := 0;
       "BMS1".BR07wAlm3 := 0;
       "BMS1".BR07wWarn1 := 0;
   ELSE
       "BMS1".BR07wAlm1 := #BR07wAlm1;
       "BMS1".BR07wAlm2 := #BR07wAlm2;
       "BMS1".BR07wAlm3 := #BR07wAlm3;
       "BMS1".BR07wWarn1 := #BR07wWarn1;
   END_IF;

   IF "HMI".xBB1BR8AlmDisable OR "HMI".xBB1AlmDisable OR "HMI".xPEMSAlmDisable OR "HMI".xPIAlmDisable
   THEN
       "BMS1".BR08wAlm1 := 0;
       "BMS1".BR08wAlm2 := 0;
       "BMS1".BR08wAlm3 := 0;
       "BMS1".BR08wWarn1 := 0;
   ELSE
       "BMS1".BR08wAlm1 := #BR08wAlm1;
       "BMS1".BR08wAlm2 := #BR08wAlm2;
       "BMS1".BR08wAlm3 := #BR08wAlm3;
       "BMS1".BR08wWarn1 := #BR08wWarn1;
   END_IF;
END_REGION

REGION Network 62: Alarm SBMU 9/10
   RUNG wire#powerrail
      "SBMU Alarm"("In Word1" := "BMS1".BR09.wWarn1, "In Word2" := "BMS1".BR09.wWarn2, "In Word3" := "BMS1".BR09.wWarn3, "In Word4" := "BMS1".BR09.wWarn4, "Out Alm1" => #BR09wAlm1, "Out Alm2" => #BR09wAlm2, "Out Alm3" => #BR09wAlm3, "Out Warn1" => #BR09wWarn1)
      "SBMU Alarm"("In Word1" := "BMS1".BR10.wWarn1, "In Word2" := "BMS1".BR10.wWarn2, "In Word3" := "BMS1".BR10.wWarn3, "In Word4" := "BMS1".BR10.wWarn4, "Out Alm1" => #BR10wAlm1, "Out Alm2" => #BR10wAlm2, "Out Alm3" => #BR10wAlm3, "Out Warn1" => #BR10wWarn1)
   END_RUNG
   // the same network as SCL:
   "SBMU Alarm"("In Word1" := "BMS1".BR09.wWarn1,
                "In Word2" := "BMS1".BR09.wWarn2,
                "In Word3" := "BMS1".BR09.wWarn3,
                "In Word4" := "BMS1".BR09.wWarn4,
                "Out Alm1" => #BR09wAlm1,
                "Out Alm2" => #BR09wAlm2,
                "Out Alm3" => #BR09wAlm3,
                "Out Warn1" => #BR09wWarn1,
                ENO => #_w1);
   IF #_w1 THEN
       "SBMU Alarm"("In Word1" := "BMS1".BR10.wWarn1,
                    "In Word2" := "BMS1".BR10.wWarn2,
                    "In Word3" := "BMS1".BR10.wWarn3,
                    "In Word4" := "BMS1".BR10.wWarn4,
                    "Out Alm1" => #BR10wAlm1,
                    "Out Alm2" => #BR10wAlm2,
                    "Out Alm3" => #BR10wAlm3,
                    "Out Warn1" => #BR10wWarn1);
   END_IF;
END_REGION

REGION Network 63 (SCL): Alarm SBMU 9/10 to HMI
   IF "HMI".xBB1BR9AlmDisable OR "HMI".xBB1AlmDisable OR "HMI".xPEMSAlmDisable OR "HMI".xPIAlmDisable
   THEN
       "BMS1".BR09wAlm1 := 0;
       "BMS1".BR09wAlm2 := 0;
       "BMS1".BR09wAlm3 := 0;
       "BMS1".BR09wWarn1 := 0;
   ELSE
       "BMS1".BR09wAlm1 := #BR09wAlm1;
       "BMS1".BR09wAlm2 := #BR09wAlm2;
       "BMS1".BR09wAlm3 := #BR09wAlm3;
       "BMS1".BR09wWarn1 := #BR09wWarn1;
   END_IF;

   IF "HMI".xBB1BR10AlmDisable OR "HMI".xBB1AlmDisable OR "HMI".xPEMSAlmDisable OR "HMI".xPIAlmDisable
   THEN
       "BMS1".BR10wAlm1 := 0;
       "BMS1".BR10wAlm2 := 0;
       "BMS1".BR10wAlm3 := 0;
       "BMS1".BR10wWarn1 := 0;
   ELSE
       "BMS1".BR10wAlm1 := #BR10wAlm1;
       "BMS1".BR10wAlm2 := #BR10wAlm2;
       "BMS1".BR10wAlm3 := #BR10wAlm3;
       "BMS1".BR10wWarn1 := #BR10wWarn1;
   END_IF;
END_REGION

REGION Network 64: Alarm SBMU 11/12
   RUNG wire#powerrail
      "SBMU Alarm"("In Word1" := "BMS1".BR11.wWarn1, "In Word2" := "BMS1".BR11.wWarn2, "In Word3" := "BMS1".BR11.wWarn3, "In Word4" := "BMS1".BR11.wWarn4, "Out Alm1" => #BR11wAlm1, "Out Alm2" => #BR11wAlm2, "Out Alm3" => #BR11wAlm3, "Out Warn1" => #BR11wWarn1)
      "SBMU Alarm"("In Word1" := "BMS1".BR12.wWarn1, "In Word2" := "BMS1".BR12.wWarn2, "In Word3" := "BMS1".BR12.wWarn3, "In Word4" := "BMS1".BR12.wWarn4, "Out Alm1" => #BR12wAlm1, "Out Alm2" => #BR12wAlm2, "Out Alm3" => #BR12wAlm3, "Out Warn1" => #BR12wWarn1)
   END_RUNG
   // the same network as SCL:
   "SBMU Alarm"("In Word1" := "BMS1".BR11.wWarn1,
                "In Word2" := "BMS1".BR11.wWarn2,
                "In Word3" := "BMS1".BR11.wWarn3,
                "In Word4" := "BMS1".BR11.wWarn4,
                "Out Alm1" => #BR11wAlm1,
                "Out Alm2" => #BR11wAlm2,
                "Out Alm3" => #BR11wAlm3,
                "Out Warn1" => #BR11wWarn1,
                ENO => #_w1);
   IF #_w1 THEN
       "SBMU Alarm"("In Word1" := "BMS1".BR12.wWarn1,
                    "In Word2" := "BMS1".BR12.wWarn2,
                    "In Word3" := "BMS1".BR12.wWarn3,
                    "In Word4" := "BMS1".BR12.wWarn4,
                    "Out Alm1" => #BR12wAlm1,
                    "Out Alm2" => #BR12wAlm2,
                    "Out Alm3" => #BR12wAlm3,
                    "Out Warn1" => #BR12wWarn1);
   END_IF;
END_REGION

REGION Network 65 (SCL): Alarm SBMU11/12 to HMI
   IF "HMI".xBB1BR11AlmDisable OR "HMI".xBB1AlmDisable OR "HMI".xPEMSAlmDisable OR "HMI".xPIAlmDisable
   THEN
       "BMS1".BR11wAlm1 := 0;
       "BMS1".BR11wAlm2 := 0;
       "BMS1".BR11wAlm3 := 0;
       "BMS1".BR11wWarn1 := 0;
   ELSE
       "BMS1".BR11wAlm1 := #BR11wAlm1;
       "BMS1".BR11wAlm2 := #BR11wAlm2;
       "BMS1".BR11wAlm3 := #BR11wAlm3;
       "BMS1".BR11wWarn1 := #BR11wWarn1;
   END_IF;

   IF "HMI".xBB1BR12AlmDisable OR "HMI".xBB1AlmDisable OR "HMI".xPEMSAlmDisable OR "HMI".xPIAlmDisable
   THEN
       "BMS1".BR12wAlm1 := 0;
       "BMS1".BR12wAlm2 := 0;
       "BMS1".BR12wAlm3 := 0;
       "BMS1".BR12wWarn1 := 0;
   ELSE
       "BMS1".BR12wAlm1 := #BR12wAlm1;
       "BMS1".BR12wAlm2 := #BR12wAlm2;
       "BMS1".BR12wAlm3 := #BR12wAlm3;
       "BMS1".BR12wWarn1 := #BR12wWarn1;
   END_IF;
END_REGION

REGION Network 67: BMS1 Fault SubSystem
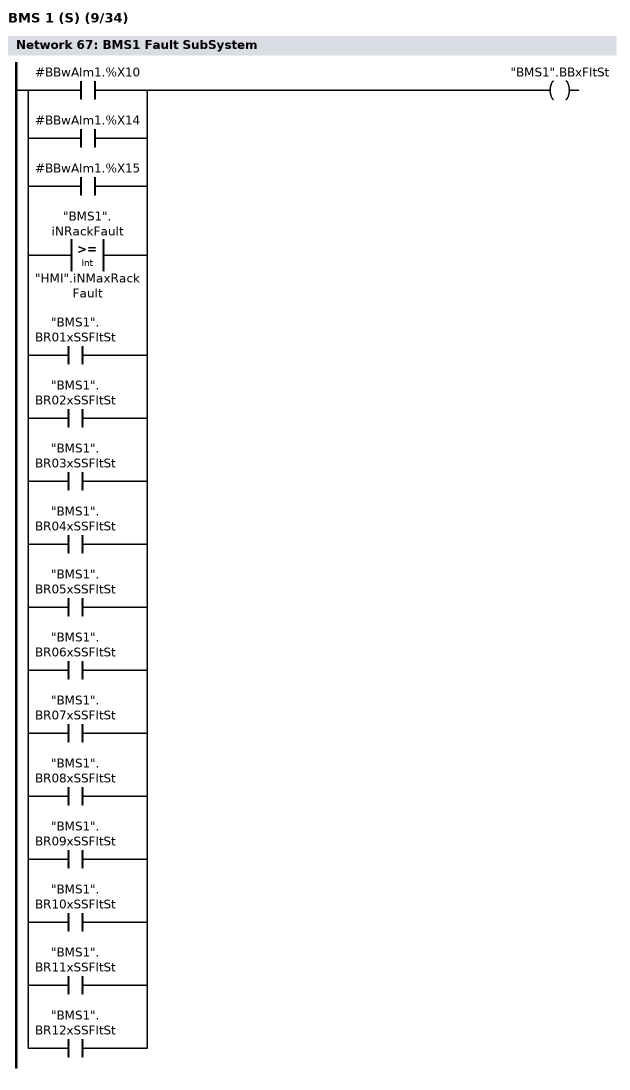
   RUNG wire#powerrail
      Contact( #BBwAlm1.%X10 )
      wire#w1
      Coil( "BMS1".BBxFltSt )
   END_RUNG
   RUNG wire#powerrail
      Contact( #BBwAlm1.%X14 )
   END_RUNG wire#w1
   RUNG wire#powerrail
      Contact( #BBwAlm1.%X15 )
   END_RUNG wire#w1
   RUNG wire#powerrail
      { S7_Templates := "SrcType := Int" } GE_Contact(in1 := "BMS1".iNRackFault, in2 := "HMI".iNMaxRackFault)
   END_RUNG wire#w1
   RUNG wire#powerrail
      Contact( "BMS1".BR01xSSFltSt )
   END_RUNG wire#w1
   RUNG wire#powerrail
      Contact( "BMS1".BR02xSSFltSt )
   END_RUNG wire#w1
   RUNG wire#powerrail
      Contact( "BMS1".BR03xSSFltSt )
   END_RUNG wire#w1
   RUNG wire#powerrail
      Contact( "BMS1".BR04xSSFltSt )
   END_RUNG wire#w1
   RUNG wire#powerrail
      Contact( "BMS1".BR05xSSFltSt )
   END_RUNG wire#w1
   RUNG wire#powerrail
      Contact( "BMS1".BR06xSSFltSt )
   END_RUNG wire#w1
   RUNG wire#powerrail
      Contact( "BMS1".BR07xSSFltSt )
   END_RUNG wire#w1
   RUNG wire#powerrail
      Contact( "BMS1".BR08xSSFltSt )
   END_RUNG wire#w1
   RUNG wire#powerrail
      Contact( "BMS1".BR09xSSFltSt )
   END_RUNG wire#w1
   RUNG wire#powerrail
      Contact( "BMS1".BR10xSSFltSt )
   END_RUNG wire#w1
   RUNG wire#powerrail
      Contact( "BMS1".BR11xSSFltSt )
   END_RUNG wire#w1
   RUNG wire#powerrail
      Contact( "BMS1".BR12xSSFltSt )
   END_RUNG wire#w1
   // the same network as SCL:
   "BMS1".BBxFltSt := #BBwAlm1.%X10 OR #BBwAlm1.%X14 OR #BBwAlm1.%X15 OR ("BMS1".iNRackFault >= "HMI".iNMaxRackFault) OR "BMS1".BR01xSSFltSt OR "BMS1".BR02xSSFltSt OR "BMS1".BR03xSSFltSt OR "BMS1".BR04xSSFltSt OR "BMS1".BR05xSSFltSt OR "BMS1".BR06xSSFltSt OR "BMS1".BR07xSSFltSt OR "BMS1".BR08xSSFltSt OR "BMS1".BR09xSSFltSt OR "BMS1".BR10xSSFltSt OR "BMS1".BR11xSSFltSt OR "BMS1".BR12xSSFltSt;
END_REGION

REGION Network 68: BMS1 Alarm
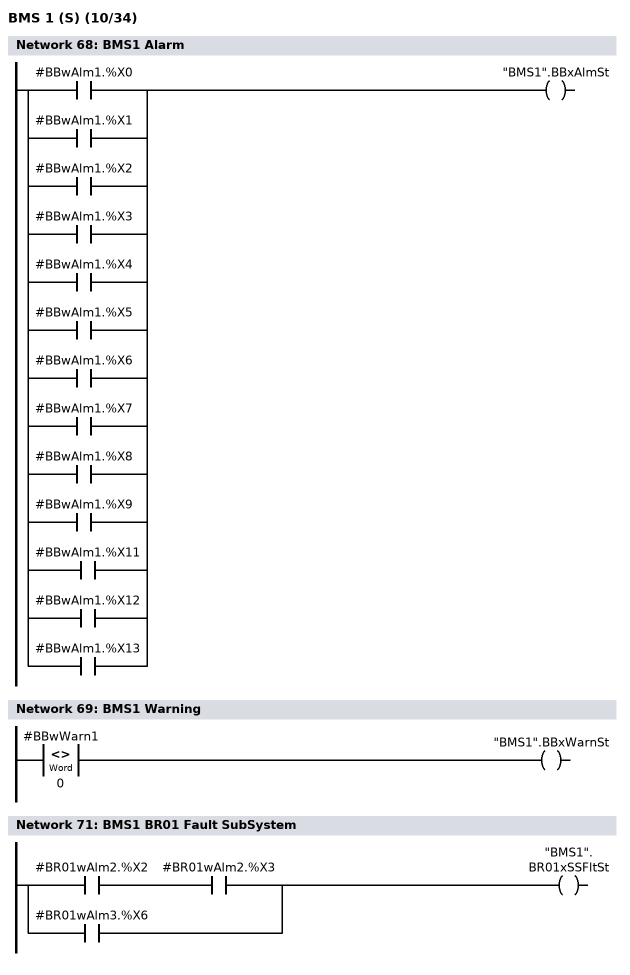
   RUNG wire#powerrail
      Contact( #BBwAlm1.%X0 )
      wire#w1
      Coil( "BMS1".BBxAlmSt )
   END_RUNG
   RUNG wire#powerrail
      Contact( #BBwAlm1.%X1 )
   END_RUNG wire#w1
   RUNG wire#powerrail
      Contact( #BBwAlm1.%X2 )
   END_RUNG wire#w1
   RUNG wire#powerrail
      Contact( #BBwAlm1.%X3 )
   END_RUNG wire#w1
   RUNG wire#powerrail
      Contact( #BBwAlm1.%X4 )
   END_RUNG wire#w1
   RUNG wire#powerrail
      Contact( #BBwAlm1.%X5 )
   END_RUNG wire#w1
   RUNG wire#powerrail
      Contact( #BBwAlm1.%X6 )
   END_RUNG wire#w1
   RUNG wire#powerrail
      Contact( #BBwAlm1.%X7 )
   END_RUNG wire#w1
   RUNG wire#powerrail
      Contact( #BBwAlm1.%X8 )
   END_RUNG wire#w1
   RUNG wire#powerrail
      Contact( #BBwAlm1.%X9 )
   END_RUNG wire#w1
   RUNG wire#powerrail
      Contact( #BBwAlm1.%X11 )
   END_RUNG wire#w1
   RUNG wire#powerrail
      Contact( #BBwAlm1.%X12 )
   END_RUNG wire#w1
   RUNG wire#powerrail
      Contact( #BBwAlm1.%X13 )
   END_RUNG wire#w1
   // the same network as SCL:
   "BMS1".BBxAlmSt := #BBwAlm1.%X0 OR #BBwAlm1.%X1 OR #BBwAlm1.%X2 OR #BBwAlm1.%X3 OR #BBwAlm1.%X4 OR #BBwAlm1.%X5 OR #BBwAlm1.%X6 OR #BBwAlm1.%X7 OR #BBwAlm1.%X8 OR #BBwAlm1.%X9 OR #BBwAlm1.%X11 OR #BBwAlm1.%X12 OR #BBwAlm1.%X13;
END_REGION

REGION Network 69: BMS1 Warning
   RUNG wire#powerrail
      { S7_Templates := "SrcType := Word" } NE_Contact(in1 := #BBwWarn1, in2 := 0)
      Coil( "BMS1".BBxWarnSt )
   END_RUNG
   // the same network as SCL:
   "BMS1".BBxWarnSt := #BBwWarn1 <> 0;
END_REGION

REGION Network 70 (SCL): Computing number of Rack in Fault
   "BMS1".iNRackFault := BOOL_TO_INT("BMS1".BR01xFltSt) +
   BOOL_TO_INT("BMS1".BR02xFltSt) +
   BOOL_TO_INT("BMS1".BR03xFltSt) +
   BOOL_TO_INT("BMS1".BR04xFltSt) +
   BOOL_TO_INT("BMS1".BR05xFltSt) +
   BOOL_TO_INT("BMS1".BR06xFltSt) +
   BOOL_TO_INT("BMS1".BR07xFltSt) +
   BOOL_TO_INT("BMS1".BR08xFltSt) +
   BOOL_TO_INT("BMS1".BR09xFltSt) +
   BOOL_TO_INT("BMS1".BR10xFltSt) +
   BOOL_TO_INT("BMS1".BR11xFltSt) +
   BOOL_TO_INT("BMS1".BR12xFltSt);
END_REGION

REGION Network 71: BMS1 BR01 Fault SubSystem
   RUNG wire#powerrail
      Contact( #BR01wAlm2.%X2 )
      Contact( #BR01wAlm2.%X3 )
      wire#w1
      Coil( "BMS1".BR01xSSFltSt )
   END_RUNG
   RUNG wire#powerrail
      Contact( #BR01wAlm3.%X6 )
   END_RUNG wire#w1
   // the same network as SCL:
   "BMS1".BR01xSSFltSt := (#BR01wAlm2.%X2 AND #BR01wAlm2.%X3) OR #BR01wAlm3.%X6;
END_REGION

REGION Network 72: BMS1 BR01 Fault
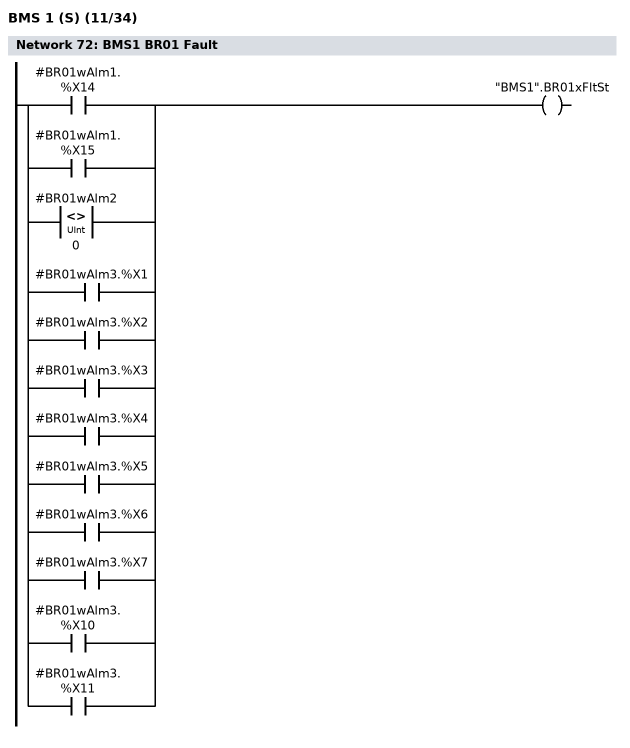
   RUNG wire#powerrail
      Contact( #BR01wAlm1.%X14 )
      wire#w1
      Coil( "BMS1".BR01xFltSt )
   END_RUNG
   RUNG wire#powerrail
      Contact( #BR01wAlm1.%X15 )
   END_RUNG wire#w1
   RUNG wire#powerrail
      { S7_Templates := "SrcType := UInt" } NE_Contact(in1 := #BR01wAlm2, in2 := 0)
   END_RUNG wire#w1
   RUNG wire#powerrail
      Contact( #BR01wAlm3.%X1 )
   END_RUNG wire#w1
   RUNG wire#powerrail
      Contact( #BR01wAlm3.%X2 )
   END_RUNG wire#w1
   RUNG wire#powerrail
      Contact( #BR01wAlm3.%X3 )
   END_RUNG wire#w1
   RUNG wire#powerrail
      Contact( #BR01wAlm3.%X4 )
   END_RUNG wire#w1
   RUNG wire#powerrail
      Contact( #BR01wAlm3.%X5 )
   END_RUNG wire#w1
   RUNG wire#powerrail
      Contact( #BR01wAlm3.%X6 )
   END_RUNG wire#w1
   RUNG wire#powerrail
      Contact( #BR01wAlm3.%X7 )
   END_RUNG wire#w1
   RUNG wire#powerrail
      Contact( #BR01wAlm3.%X10 )
   END_RUNG wire#w1
   RUNG wire#powerrail
      Contact( #BR01wAlm3.%X11 )
   END_RUNG wire#w1
   // the same network as SCL:
   "BMS1".BR01xFltSt := #BR01wAlm1.%X14 OR #BR01wAlm1.%X15 OR (#BR01wAlm2 <> 0) OR #BR01wAlm3.%X1 OR #BR01wAlm3.%X2 OR #BR01wAlm3.%X3 OR #BR01wAlm3.%X4 OR #BR01wAlm3.%X5 OR #BR01wAlm3.%X6 OR #BR01wAlm3.%X7 OR #BR01wAlm3.%X10 OR #BR01wAlm3.%X11;
END_REGION

REGION Network 73: BMS1 BR01 Alarm
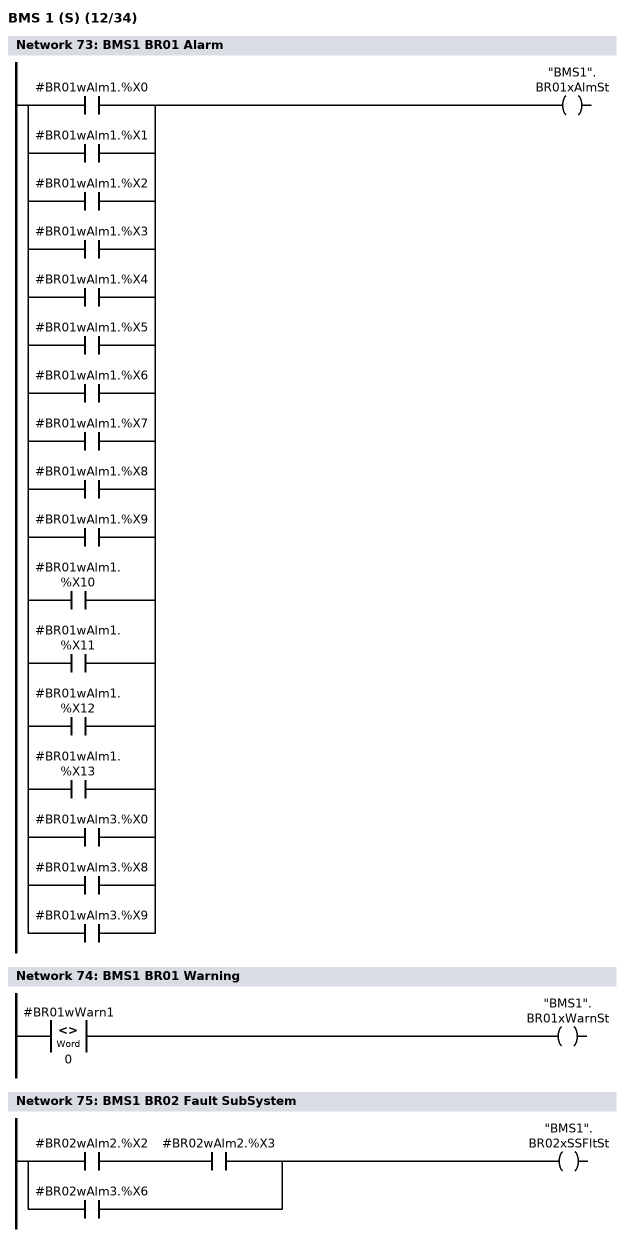
   RUNG wire#powerrail
      Contact( #BR01wAlm1.%X0 )
      wire#w1
      Coil( "BMS1".BR01xAlmSt )
   END_RUNG
   RUNG wire#powerrail
      Contact( #BR01wAlm1.%X1 )
   END_RUNG wire#w1
   RUNG wire#powerrail
      Contact( #BR01wAlm1.%X2 )
   END_RUNG wire#w1
   RUNG wire#powerrail
      Contact( #BR01wAlm1.%X3 )
   END_RUNG wire#w1
   RUNG wire#powerrail
      Contact( #BR01wAlm1.%X4 )
   END_RUNG wire#w1
   RUNG wire#powerrail
      Contact( #BR01wAlm1.%X5 )
   END_RUNG wire#w1
   RUNG wire#powerrail
      Contact( #BR01wAlm1.%X6 )
   END_RUNG wire#w1
   RUNG wire#powerrail
      Contact( #BR01wAlm1.%X7 )
   END_RUNG wire#w1
   RUNG wire#powerrail
      Contact( #BR01wAlm1.%X8 )
   END_RUNG wire#w1
   RUNG wire#powerrail
      Contact( #BR01wAlm1.%X9 )
   END_RUNG wire#w1
   RUNG wire#powerrail
      Contact( #BR01wAlm1.%X10 )
   END_RUNG wire#w1
   RUNG wire#powerrail
      Contact( #BR01wAlm1.%X11 )
   END_RUNG wire#w1
   RUNG wire#powerrail
      Contact( #BR01wAlm1.%X12 )
   END_RUNG wire#w1
   RUNG wire#powerrail
      Contact( #BR01wAlm1.%X13 )
   END_RUNG wire#w1
   RUNG wire#powerrail
      Contact( #BR01wAlm3.%X0 )
   END_RUNG wire#w1
   RUNG wire#powerrail
      Contact( #BR01wAlm3.%X8 )
   END_RUNG wire#w1
   RUNG wire#powerrail
      Contact( #BR01wAlm3.%X9 )
   END_RUNG wire#w1
   // the same network as SCL:
   "BMS1".BR01xAlmSt := #BR01wAlm1.%X0 OR #BR01wAlm1.%X1 OR #BR01wAlm1.%X2 OR #BR01wAlm1.%X3 OR #BR01wAlm1.%X4 OR #BR01wAlm1.%X5 OR #BR01wAlm1.%X6 OR #BR01wAlm1.%X7 OR #BR01wAlm1.%X8 OR #BR01wAlm1.%X9 OR #BR01wAlm1.%X10 OR #BR01wAlm1.%X11 OR #BR01wAlm1.%X12 OR #BR01wAlm1.%X13 OR #BR01wAlm3.%X0 OR #BR01wAlm3.%X8 OR #BR01wAlm3.%X9;
END_REGION

REGION Network 74: BMS1 BR01 Warning
   RUNG wire#powerrail
      { S7_Templates := "SrcType := Word" } NE_Contact(in1 := #BR01wWarn1, in2 := 0)
      Coil( "BMS1".BR01xWarnSt )
   END_RUNG
   // the same network as SCL:
   "BMS1".BR01xWarnSt := #BR01wWarn1 <> 0;
END_REGION

REGION Network 75: BMS1 BR02 Fault SubSystem
   RUNG wire#powerrail
      Contact( #BR02wAlm2.%X2 )
      Contact( #BR02wAlm2.%X3 )
      wire#w1
      Coil( "BMS1".BR02xSSFltSt )
   END_RUNG
   RUNG wire#powerrail
      Contact( #BR02wAlm3.%X6 )
   END_RUNG wire#w1
   // the same network as SCL:
   "BMS1".BR02xSSFltSt := (#BR02wAlm2.%X2 AND #BR02wAlm2.%X3) OR #BR02wAlm3.%X6;
END_REGION

REGION Network 76: BMS1 BR02 Fault
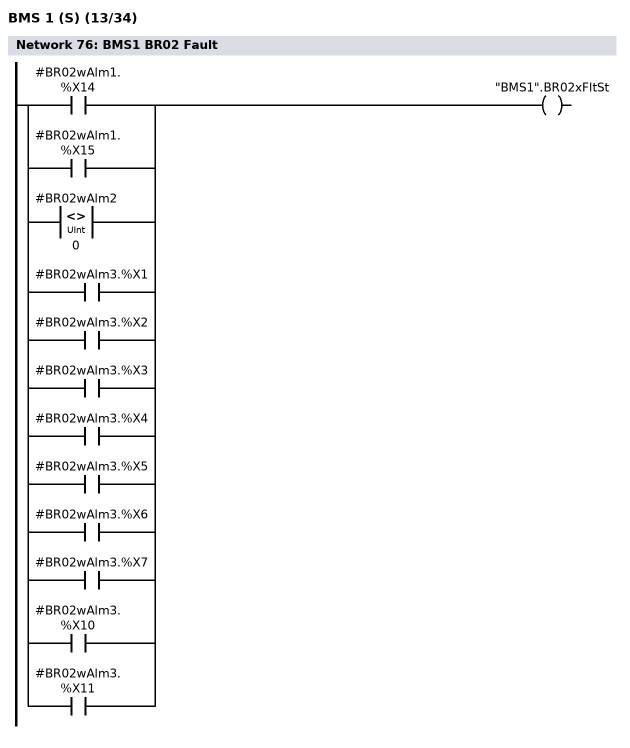
   RUNG wire#powerrail
      Contact( #BR02wAlm1.%X14 )
      wire#w1
      Coil( "BMS1".BR02xFltSt )
   END_RUNG
   RUNG wire#powerrail
      Contact( #BR02wAlm1.%X15 )
   END_RUNG wire#w1
   RUNG wire#powerrail
      { S7_Templates := "SrcType := UInt" } NE_Contact(in1 := #BR02wAlm2, in2 := 0)
   END_RUNG wire#w1
   RUNG wire#powerrail
      Contact( #BR02wAlm3.%X1 )
   END_RUNG wire#w1
   RUNG wire#powerrail
      Contact( #BR02wAlm3.%X2 )
   END_RUNG wire#w1
   RUNG wire#powerrail
      Contact( #BR02wAlm3.%X3 )
   END_RUNG wire#w1
   RUNG wire#powerrail
      Contact( #BR02wAlm3.%X4 )
   END_RUNG wire#w1
   RUNG wire#powerrail
      Contact( #BR02wAlm3.%X5 )
   END_RUNG wire#w1
   RUNG wire#powerrail
      Contact( #BR02wAlm3.%X6 )
   END_RUNG wire#w1
   RUNG wire#powerrail
      Contact( #BR02wAlm3.%X7 )
   END_RUNG wire#w1
   RUNG wire#powerrail
      Contact( #BR02wAlm3.%X10 )
   END_RUNG wire#w1
   RUNG wire#powerrail
      Contact( #BR02wAlm3.%X11 )
   END_RUNG wire#w1
   // the same network as SCL:
   "BMS1".BR02xFltSt := #BR02wAlm1.%X14 OR #BR02wAlm1.%X15 OR (#BR02wAlm2 <> 0) OR #BR02wAlm3.%X1 OR #BR02wAlm3.%X2 OR #BR02wAlm3.%X3 OR #BR02wAlm3.%X4 OR #BR02wAlm3.%X5 OR #BR02wAlm3.%X6 OR #BR02wAlm3.%X7 OR #BR02wAlm3.%X10 OR #BR02wAlm3.%X11;
END_REGION

REGION Network 77: BMS1 BR02 Alarm
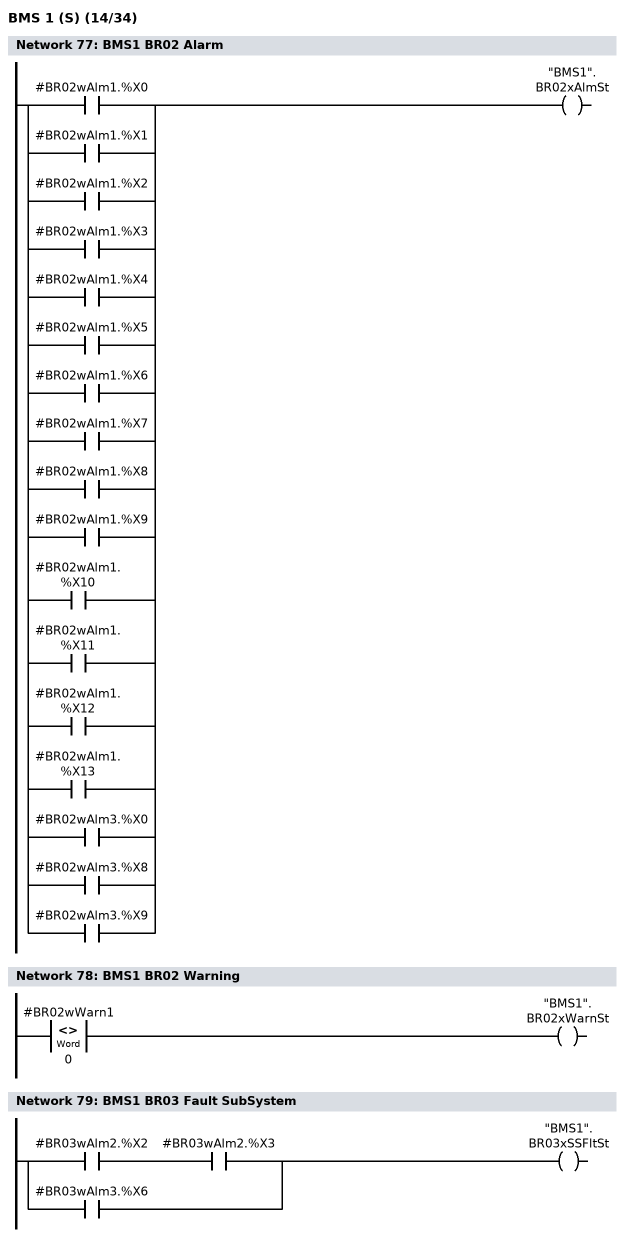
   RUNG wire#powerrail
      Contact( #BR02wAlm1.%X0 )
      wire#w1
      Coil( "BMS1".BR02xAlmSt )
   END_RUNG
   RUNG wire#powerrail
      Contact( #BR02wAlm1.%X1 )
   END_RUNG wire#w1
   RUNG wire#powerrail
      Contact( #BR02wAlm1.%X2 )
   END_RUNG wire#w1
   RUNG wire#powerrail
      Contact( #BR02wAlm1.%X3 )
   END_RUNG wire#w1
   RUNG wire#powerrail
      Contact( #BR02wAlm1.%X4 )
   END_RUNG wire#w1
   RUNG wire#powerrail
      Contact( #BR02wAlm1.%X5 )
   END_RUNG wire#w1
   RUNG wire#powerrail
      Contact( #BR02wAlm1.%X6 )
   END_RUNG wire#w1
   RUNG wire#powerrail
      Contact( #BR02wAlm1.%X7 )
   END_RUNG wire#w1
   RUNG wire#powerrail
      Contact( #BR02wAlm1.%X8 )
   END_RUNG wire#w1
   RUNG wire#powerrail
      Contact( #BR02wAlm1.%X9 )
   END_RUNG wire#w1
   RUNG wire#powerrail
      Contact( #BR02wAlm1.%X10 )
   END_RUNG wire#w1
   RUNG wire#powerrail
      Contact( #BR02wAlm1.%X11 )
   END_RUNG wire#w1
   RUNG wire#powerrail
      Contact( #BR02wAlm1.%X12 )
   END_RUNG wire#w1
   RUNG wire#powerrail
      Contact( #BR02wAlm1.%X13 )
   END_RUNG wire#w1
   RUNG wire#powerrail
      Contact( #BR02wAlm3.%X0 )
   END_RUNG wire#w1
   RUNG wire#powerrail
      Contact( #BR02wAlm3.%X8 )
   END_RUNG wire#w1
   RUNG wire#powerrail
      Contact( #BR02wAlm3.%X9 )
   END_RUNG wire#w1
   // the same network as SCL:
   "BMS1".BR02xAlmSt := #BR02wAlm1.%X0 OR #BR02wAlm1.%X1 OR #BR02wAlm1.%X2 OR #BR02wAlm1.%X3 OR #BR02wAlm1.%X4 OR #BR02wAlm1.%X5 OR #BR02wAlm1.%X6 OR #BR02wAlm1.%X7 OR #BR02wAlm1.%X8 OR #BR02wAlm1.%X9 OR #BR02wAlm1.%X10 OR #BR02wAlm1.%X11 OR #BR02wAlm1.%X12 OR #BR02wAlm1.%X13 OR #BR02wAlm3.%X0 OR #BR02wAlm3.%X8 OR #BR02wAlm3.%X9;
END_REGION

REGION Network 78: BMS1 BR02 Warning
   RUNG wire#powerrail
      { S7_Templates := "SrcType := Word" } NE_Contact(in1 := #BR02wWarn1, in2 := 0)
      Coil( "BMS1".BR02xWarnSt )
   END_RUNG
   // the same network as SCL:
   "BMS1".BR02xWarnSt := #BR02wWarn1 <> 0;
END_REGION

REGION Network 79: BMS1 BR03 Fault SubSystem
   RUNG wire#powerrail
      Contact( #BR03wAlm2.%X2 )
      Contact( #BR03wAlm2.%X3 )
      wire#w1
      Coil( "BMS1".BR03xSSFltSt )
   END_RUNG
   RUNG wire#powerrail
      Contact( #BR03wAlm3.%X6 )
   END_RUNG wire#w1
   // the same network as SCL:
   "BMS1".BR03xSSFltSt := (#BR03wAlm2.%X2 AND #BR03wAlm2.%X3) OR #BR03wAlm3.%X6;
END_REGION

REGION Network 80: BMS1 BR03 Fault
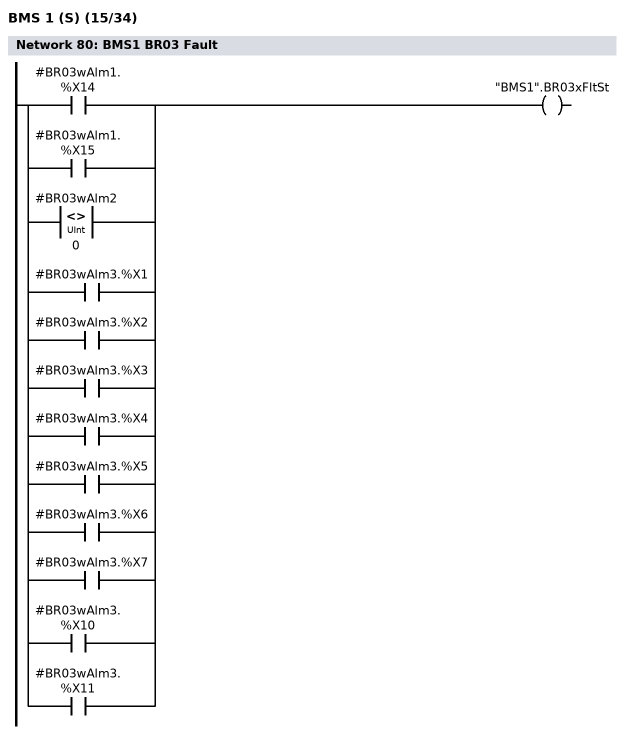
   RUNG wire#powerrail
      Contact( #BR03wAlm1.%X14 )
      wire#w1
      Coil( "BMS1".BR03xFltSt )
   END_RUNG
   RUNG wire#powerrail
      Contact( #BR03wAlm1.%X15 )
   END_RUNG wire#w1
   RUNG wire#powerrail
      { S7_Templates := "SrcType := UInt" } NE_Contact(in1 := #BR03wAlm2, in2 := 0)
   END_RUNG wire#w1
   RUNG wire#powerrail
      Contact( #BR03wAlm3.%X1 )
   END_RUNG wire#w1
   RUNG wire#powerrail
      Contact( #BR03wAlm3.%X2 )
   END_RUNG wire#w1
   RUNG wire#powerrail
      Contact( #BR03wAlm3.%X3 )
   END_RUNG wire#w1
   RUNG wire#powerrail
      Contact( #BR03wAlm3.%X4 )
   END_RUNG wire#w1
   RUNG wire#powerrail
      Contact( #BR03wAlm3.%X5 )
   END_RUNG wire#w1
   RUNG wire#powerrail
      Contact( #BR03wAlm3.%X6 )
   END_RUNG wire#w1
   RUNG wire#powerrail
      Contact( #BR03wAlm3.%X7 )
   END_RUNG wire#w1
   RUNG wire#powerrail
      Contact( #BR03wAlm3.%X10 )
   END_RUNG wire#w1
   RUNG wire#powerrail
      Contact( #BR03wAlm3.%X11 )
   END_RUNG wire#w1
   // the same network as SCL:
   "BMS1".BR03xFltSt := #BR03wAlm1.%X14 OR #BR03wAlm1.%X15 OR (#BR03wAlm2 <> 0) OR #BR03wAlm3.%X1 OR #BR03wAlm3.%X2 OR #BR03wAlm3.%X3 OR #BR03wAlm3.%X4 OR #BR03wAlm3.%X5 OR #BR03wAlm3.%X6 OR #BR03wAlm3.%X7 OR #BR03wAlm3.%X10 OR #BR03wAlm3.%X11;
END_REGION

REGION Network 81: BMS1 BR03 Alarm
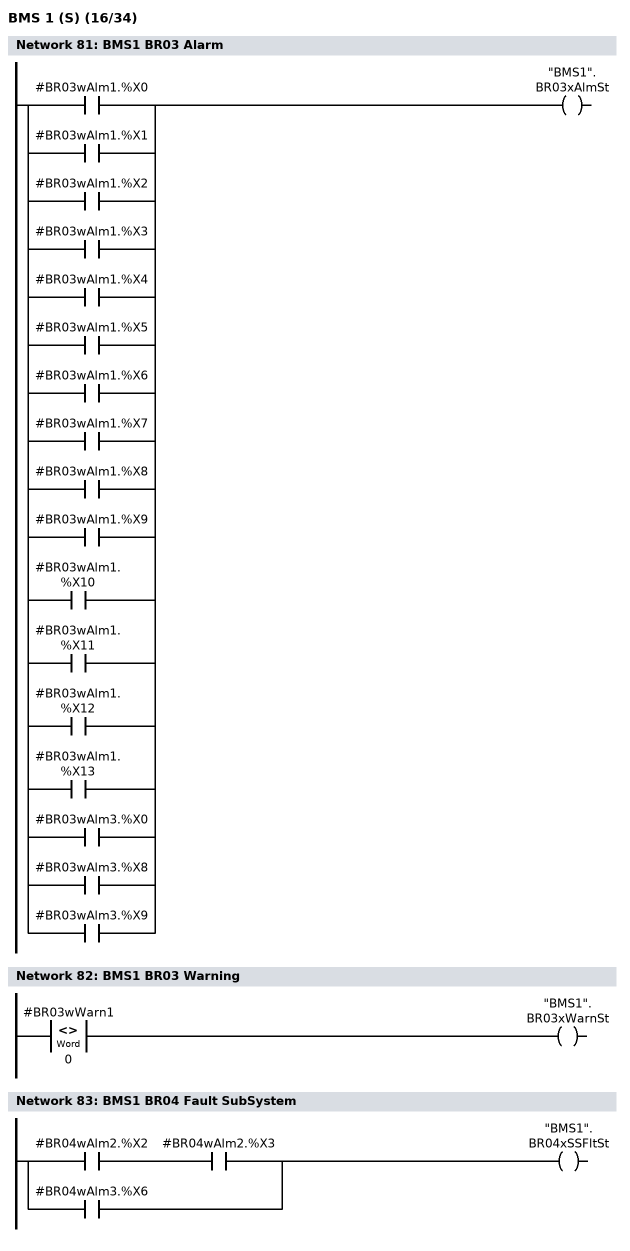
   RUNG wire#powerrail
      Contact( #BR03wAlm1.%X0 )
      wire#w1
      Coil( "BMS1".BR03xAlmSt )
   END_RUNG
   RUNG wire#powerrail
      Contact( #BR03wAlm1.%X1 )
   END_RUNG wire#w1
   RUNG wire#powerrail
      Contact( #BR03wAlm1.%X2 )
   END_RUNG wire#w1
   RUNG wire#powerrail
      Contact( #BR03wAlm1.%X3 )
   END_RUNG wire#w1
   RUNG wire#powerrail
      Contact( #BR03wAlm1.%X4 )
   END_RUNG wire#w1
   RUNG wire#powerrail
      Contact( #BR03wAlm1.%X5 )
   END_RUNG wire#w1
   RUNG wire#powerrail
      Contact( #BR03wAlm1.%X6 )
   END_RUNG wire#w1
   RUNG wire#powerrail
      Contact( #BR03wAlm1.%X7 )
   END_RUNG wire#w1
   RUNG wire#powerrail
      Contact( #BR03wAlm1.%X8 )
   END_RUNG wire#w1
   RUNG wire#powerrail
      Contact( #BR03wAlm1.%X9 )
   END_RUNG wire#w1
   RUNG wire#powerrail
      Contact( #BR03wAlm1.%X10 )
   END_RUNG wire#w1
   RUNG wire#powerrail
      Contact( #BR03wAlm1.%X11 )
   END_RUNG wire#w1
   RUNG wire#powerrail
      Contact( #BR03wAlm1.%X12 )
   END_RUNG wire#w1
   RUNG wire#powerrail
      Contact( #BR03wAlm1.%X13 )
   END_RUNG wire#w1
   RUNG wire#powerrail
      Contact( #BR03wAlm3.%X0 )
   END_RUNG wire#w1
   RUNG wire#powerrail
      Contact( #BR03wAlm3.%X8 )
   END_RUNG wire#w1
   RUNG wire#powerrail
      Contact( #BR03wAlm3.%X9 )
   END_RUNG wire#w1
   // the same network as SCL:
   "BMS1".BR03xAlmSt := #BR03wAlm1.%X0 OR #BR03wAlm1.%X1 OR #BR03wAlm1.%X2 OR #BR03wAlm1.%X3 OR #BR03wAlm1.%X4 OR #BR03wAlm1.%X5 OR #BR03wAlm1.%X6 OR #BR03wAlm1.%X7 OR #BR03wAlm1.%X8 OR #BR03wAlm1.%X9 OR #BR03wAlm1.%X10 OR #BR03wAlm1.%X11 OR #BR03wAlm1.%X12 OR #BR03wAlm1.%X13 OR #BR03wAlm3.%X0 OR #BR03wAlm3.%X8 OR #BR03wAlm3.%X9;
END_REGION

REGION Network 82: BMS1 BR03 Warning
   RUNG wire#powerrail
      { S7_Templates := "SrcType := Word" } NE_Contact(in1 := #BR03wWarn1, in2 := 0)
      Coil( "BMS1".BR03xWarnSt )
   END_RUNG
   // the same network as SCL:
   "BMS1".BR03xWarnSt := #BR03wWarn1 <> 0;
END_REGION

REGION Network 83: BMS1 BR04 Fault SubSystem
   RUNG wire#powerrail
      Contact( #BR04wAlm2.%X2 )
      Contact( #BR04wAlm2.%X3 )
      wire#w1
      Coil( "BMS1".BR04xSSFltSt )
   END_RUNG
   RUNG wire#powerrail
      Contact( #BR04wAlm3.%X6 )
   END_RUNG wire#w1
   // the same network as SCL:
   "BMS1".BR04xSSFltSt := (#BR04wAlm2.%X2 AND #BR04wAlm2.%X3) OR #BR04wAlm3.%X6;
END_REGION

REGION Network 84: BMS1 BR04 Fault
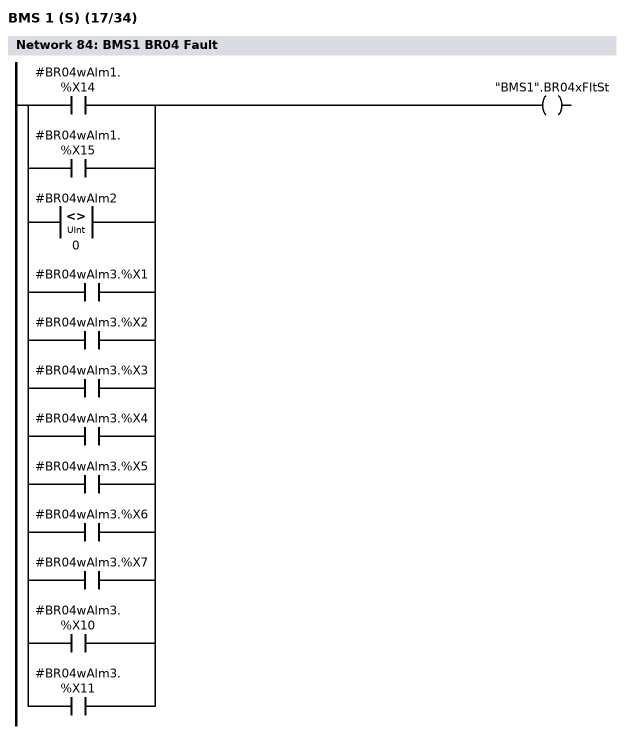
   RUNG wire#powerrail
      Contact( #BR04wAlm1.%X14 )
      wire#w1
      Coil( "BMS1".BR04xFltSt )
   END_RUNG
   RUNG wire#powerrail
      Contact( #BR04wAlm1.%X15 )
   END_RUNG wire#w1
   RUNG wire#powerrail
      { S7_Templates := "SrcType := UInt" } NE_Contact(in1 := #BR04wAlm2, in2 := 0)
   END_RUNG wire#w1
   RUNG wire#powerrail
      Contact( #BR04wAlm3.%X1 )
   END_RUNG wire#w1
   RUNG wire#powerrail
      Contact( #BR04wAlm3.%X2 )
   END_RUNG wire#w1
   RUNG wire#powerrail
      Contact( #BR04wAlm3.%X3 )
   END_RUNG wire#w1
   RUNG wire#powerrail
      Contact( #BR04wAlm3.%X4 )
   END_RUNG wire#w1
   RUNG wire#powerrail
      Contact( #BR04wAlm3.%X5 )
   END_RUNG wire#w1
   RUNG wire#powerrail
      Contact( #BR04wAlm3.%X6 )
   END_RUNG wire#w1
   RUNG wire#powerrail
      Contact( #BR04wAlm3.%X7 )
   END_RUNG wire#w1
   RUNG wire#powerrail
      Contact( #BR04wAlm3.%X10 )
   END_RUNG wire#w1
   RUNG wire#powerrail
      Contact( #BR04wAlm3.%X11 )
   END_RUNG wire#w1
   // the same network as SCL:
   "BMS1".BR04xFltSt := #BR04wAlm1.%X14 OR #BR04wAlm1.%X15 OR (#BR04wAlm2 <> 0) OR #BR04wAlm3.%X1 OR #BR04wAlm3.%X2 OR #BR04wAlm3.%X3 OR #BR04wAlm3.%X4 OR #BR04wAlm3.%X5 OR #BR04wAlm3.%X6 OR #BR04wAlm3.%X7 OR #BR04wAlm3.%X10 OR #BR04wAlm3.%X11;
END_REGION

REGION Network 85: BMS1 BR04 Alarm
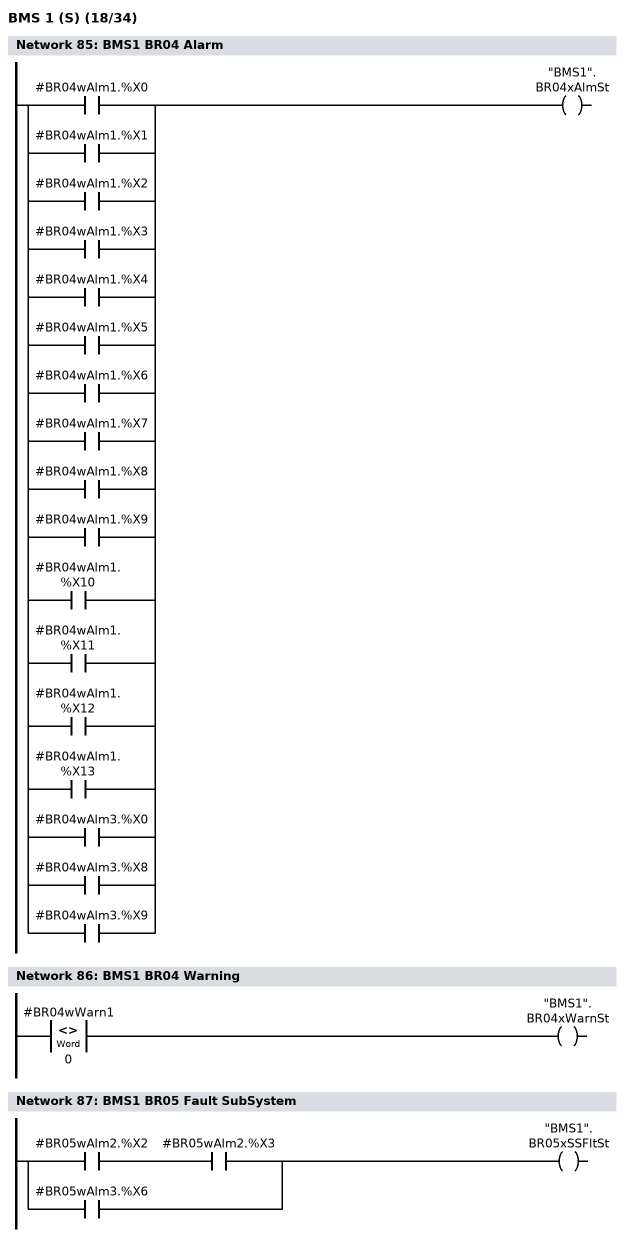
   RUNG wire#powerrail
      Contact( #BR04wAlm1.%X0 )
      wire#w1
      Coil( "BMS1".BR04xAlmSt )
   END_RUNG
   RUNG wire#powerrail
      Contact( #BR04wAlm1.%X1 )
   END_RUNG wire#w1
   RUNG wire#powerrail
      Contact( #BR04wAlm1.%X2 )
   END_RUNG wire#w1
   RUNG wire#powerrail
      Contact( #BR04wAlm1.%X3 )
   END_RUNG wire#w1
   RUNG wire#powerrail
      Contact( #BR04wAlm1.%X4 )
   END_RUNG wire#w1
   RUNG wire#powerrail
      Contact( #BR04wAlm1.%X5 )
   END_RUNG wire#w1
   RUNG wire#powerrail
      Contact( #BR04wAlm1.%X6 )
   END_RUNG wire#w1
   RUNG wire#powerrail
      Contact( #BR04wAlm1.%X7 )
   END_RUNG wire#w1
   RUNG wire#powerrail
      Contact( #BR04wAlm1.%X8 )
   END_RUNG wire#w1
   RUNG wire#powerrail
      Contact( #BR04wAlm1.%X9 )
   END_RUNG wire#w1
   RUNG wire#powerrail
      Contact( #BR04wAlm1.%X10 )
   END_RUNG wire#w1
   RUNG wire#powerrail
      Contact( #BR04wAlm1.%X11 )
   END_RUNG wire#w1
   RUNG wire#powerrail
      Contact( #BR04wAlm1.%X12 )
   END_RUNG wire#w1
   RUNG wire#powerrail
      Contact( #BR04wAlm1.%X13 )
   END_RUNG wire#w1
   RUNG wire#powerrail
      Contact( #BR04wAlm3.%X0 )
   END_RUNG wire#w1
   RUNG wire#powerrail
      Contact( #BR04wAlm3.%X8 )
   END_RUNG wire#w1
   RUNG wire#powerrail
      Contact( #BR04wAlm3.%X9 )
   END_RUNG wire#w1
   // the same network as SCL:
   "BMS1".BR04xAlmSt := #BR04wAlm1.%X0 OR #BR04wAlm1.%X1 OR #BR04wAlm1.%X2 OR #BR04wAlm1.%X3 OR #BR04wAlm1.%X4 OR #BR04wAlm1.%X5 OR #BR04wAlm1.%X6 OR #BR04wAlm1.%X7 OR #BR04wAlm1.%X8 OR #BR04wAlm1.%X9 OR #BR04wAlm1.%X10 OR #BR04wAlm1.%X11 OR #BR04wAlm1.%X12 OR #BR04wAlm1.%X13 OR #BR04wAlm3.%X0 OR #BR04wAlm3.%X8 OR #BR04wAlm3.%X9;
END_REGION

REGION Network 86: BMS1 BR04 Warning
   RUNG wire#powerrail
      { S7_Templates := "SrcType := Word" } NE_Contact(in1 := #BR04wWarn1, in2 := 0)
      Coil( "BMS1".BR04xWarnSt )
   END_RUNG
   // the same network as SCL:
   "BMS1".BR04xWarnSt := #BR04wWarn1 <> 0;
END_REGION

REGION Network 87: BMS1 BR05 Fault SubSystem
   RUNG wire#powerrail
      Contact( #BR05wAlm2.%X2 )
      Contact( #BR05wAlm2.%X3 )
      wire#w1
      Coil( "BMS1".BR05xSSFltSt )
   END_RUNG
   RUNG wire#powerrail
      Contact( #BR05wAlm3.%X6 )
   END_RUNG wire#w1
   // the same network as SCL:
   "BMS1".BR05xSSFltSt := (#BR05wAlm2.%X2 AND #BR05wAlm2.%X3) OR #BR05wAlm3.%X6;
END_REGION

REGION Network 88: BMS1 BR05 Fault
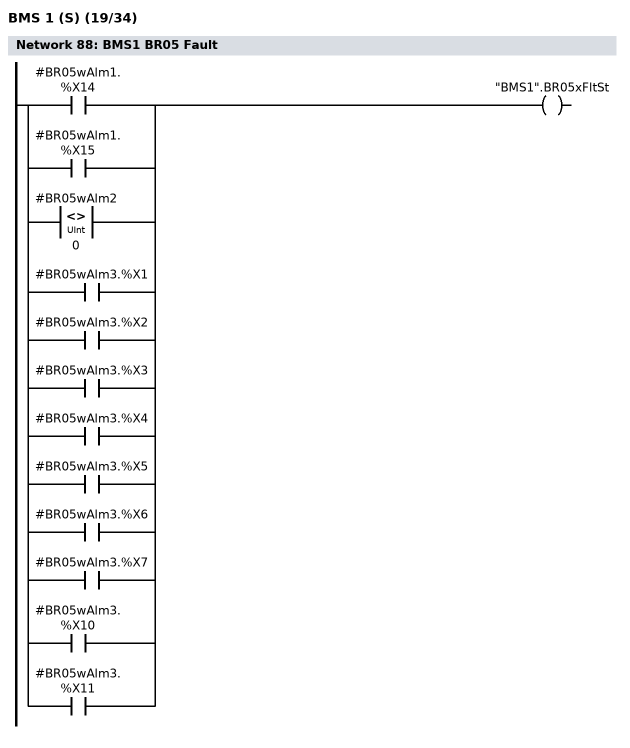
   RUNG wire#powerrail
      Contact( #BR05wAlm1.%X14 )
      wire#w1
      Coil( "BMS1".BR05xFltSt )
   END_RUNG
   RUNG wire#powerrail
      Contact( #BR05wAlm1.%X15 )
   END_RUNG wire#w1
   RUNG wire#powerrail
      { S7_Templates := "SrcType := UInt" } NE_Contact(in1 := #BR05wAlm2, in2 := 0)
   END_RUNG wire#w1
   RUNG wire#powerrail
      Contact( #BR05wAlm3.%X1 )
   END_RUNG wire#w1
   RUNG wire#powerrail
      Contact( #BR05wAlm3.%X2 )
   END_RUNG wire#w1
   RUNG wire#powerrail
      Contact( #BR05wAlm3.%X3 )
   END_RUNG wire#w1
   RUNG wire#powerrail
      Contact( #BR05wAlm3.%X4 )
   END_RUNG wire#w1
   RUNG wire#powerrail
      Contact( #BR05wAlm3.%X5 )
   END_RUNG wire#w1
   RUNG wire#powerrail
      Contact( #BR05wAlm3.%X6 )
   END_RUNG wire#w1
   RUNG wire#powerrail
      Contact( #BR05wAlm3.%X7 )
   END_RUNG wire#w1
   RUNG wire#powerrail
      Contact( #BR05wAlm3.%X10 )
   END_RUNG wire#w1
   RUNG wire#powerrail
      Contact( #BR05wAlm3.%X11 )
   END_RUNG wire#w1
   // the same network as SCL:
   "BMS1".BR05xFltSt := #BR05wAlm1.%X14 OR #BR05wAlm1.%X15 OR (#BR05wAlm2 <> 0) OR #BR05wAlm3.%X1 OR #BR05wAlm3.%X2 OR #BR05wAlm3.%X3 OR #BR05wAlm3.%X4 OR #BR05wAlm3.%X5 OR #BR05wAlm3.%X6 OR #BR05wAlm3.%X7 OR #BR05wAlm3.%X10 OR #BR05wAlm3.%X11;
END_REGION

REGION Network 89: BMS1 BR05 Alarm
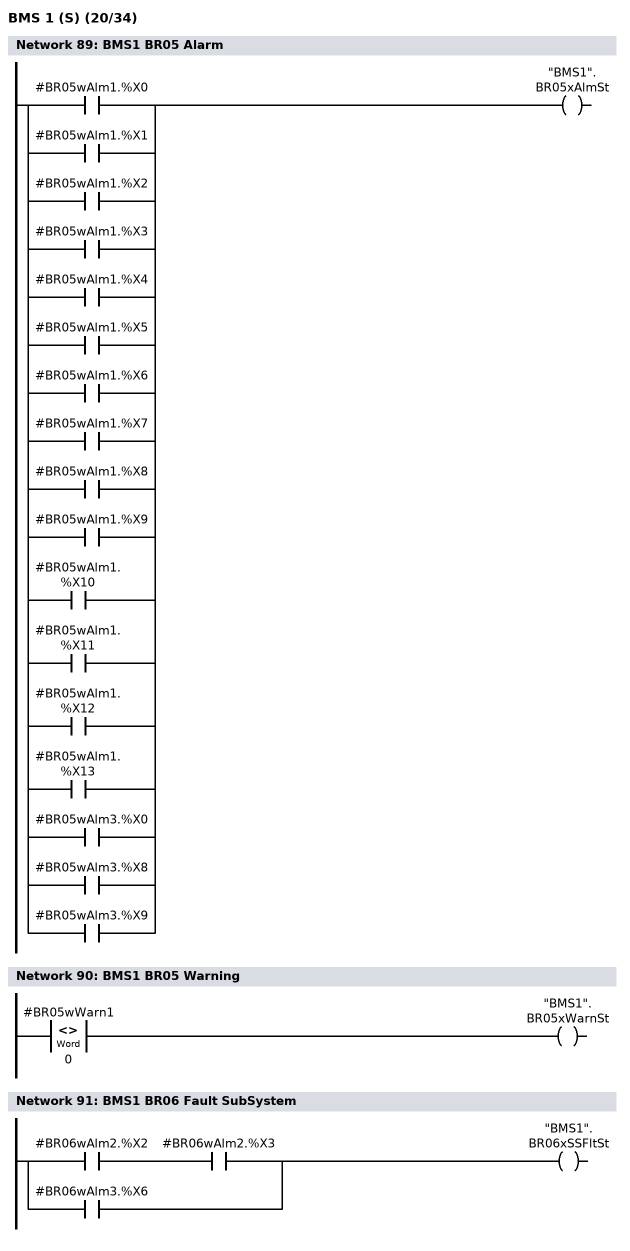
   RUNG wire#powerrail
      Contact( #BR05wAlm1.%X0 )
      wire#w1
      Coil( "BMS1".BR05xAlmSt )
   END_RUNG
   RUNG wire#powerrail
      Contact( #BR05wAlm1.%X1 )
   END_RUNG wire#w1
   RUNG wire#powerrail
      Contact( #BR05wAlm1.%X2 )
   END_RUNG wire#w1
   RUNG wire#powerrail
      Contact( #BR05wAlm1.%X3 )
   END_RUNG wire#w1
   RUNG wire#powerrail
      Contact( #BR05wAlm1.%X4 )
   END_RUNG wire#w1
   RUNG wire#powerrail
      Contact( #BR05wAlm1.%X5 )
   END_RUNG wire#w1
   RUNG wire#powerrail
      Contact( #BR05wAlm1.%X6 )
   END_RUNG wire#w1
   RUNG wire#powerrail
      Contact( #BR05wAlm1.%X7 )
   END_RUNG wire#w1
   RUNG wire#powerrail
      Contact( #BR05wAlm1.%X8 )
   END_RUNG wire#w1
   RUNG wire#powerrail
      Contact( #BR05wAlm1.%X9 )
   END_RUNG wire#w1
   RUNG wire#powerrail
      Contact( #BR05wAlm1.%X10 )
   END_RUNG wire#w1
   RUNG wire#powerrail
      Contact( #BR05wAlm1.%X11 )
   END_RUNG wire#w1
   RUNG wire#powerrail
      Contact( #BR05wAlm1.%X12 )
   END_RUNG wire#w1
   RUNG wire#powerrail
      Contact( #BR05wAlm1.%X13 )
   END_RUNG wire#w1
   RUNG wire#powerrail
      Contact( #BR05wAlm3.%X0 )
   END_RUNG wire#w1
   RUNG wire#powerrail
      Contact( #BR05wAlm3.%X8 )
   END_RUNG wire#w1
   RUNG wire#powerrail
      Contact( #BR05wAlm3.%X9 )
   END_RUNG wire#w1
   // the same network as SCL:
   "BMS1".BR05xAlmSt := #BR05wAlm1.%X0 OR #BR05wAlm1.%X1 OR #BR05wAlm1.%X2 OR #BR05wAlm1.%X3 OR #BR05wAlm1.%X4 OR #BR05wAlm1.%X5 OR #BR05wAlm1.%X6 OR #BR05wAlm1.%X7 OR #BR05wAlm1.%X8 OR #BR05wAlm1.%X9 OR #BR05wAlm1.%X10 OR #BR05wAlm1.%X11 OR #BR05wAlm1.%X12 OR #BR05wAlm1.%X13 OR #BR05wAlm3.%X0 OR #BR05wAlm3.%X8 OR #BR05wAlm3.%X9;
END_REGION

REGION Network 90: BMS1 BR05 Warning
   RUNG wire#powerrail
      { S7_Templates := "SrcType := Word" } NE_Contact(in1 := #BR05wWarn1, in2 := 0)
      Coil( "BMS1".BR05xWarnSt )
   END_RUNG
   // the same network as SCL:
   "BMS1".BR05xWarnSt := #BR05wWarn1 <> 0;
END_REGION

REGION Network 91: BMS1 BR06 Fault SubSystem
   RUNG wire#powerrail
      Contact( #BR06wAlm2.%X2 )
      Contact( #BR06wAlm2.%X3 )
      wire#w1
      Coil( "BMS1".BR06xSSFltSt )
   END_RUNG
   RUNG wire#powerrail
      Contact( #BR06wAlm3.%X6 )
   END_RUNG wire#w1
   // the same network as SCL:
   "BMS1".BR06xSSFltSt := (#BR06wAlm2.%X2 AND #BR06wAlm2.%X3) OR #BR06wAlm3.%X6;
END_REGION

REGION Network 92: BMS1 BR06 Fault
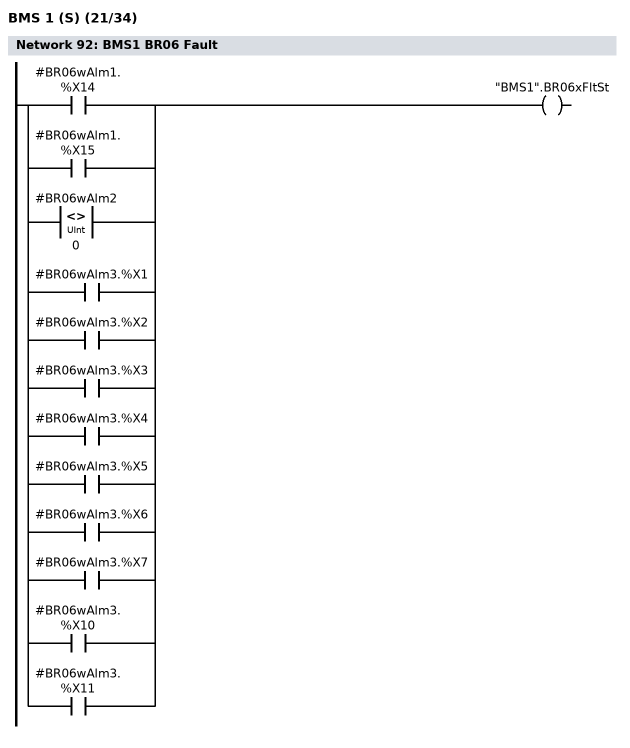
   RUNG wire#powerrail
      Contact( #BR06wAlm1.%X14 )
      wire#w1
      Coil( "BMS1".BR06xFltSt )
   END_RUNG
   RUNG wire#powerrail
      Contact( #BR06wAlm1.%X15 )
   END_RUNG wire#w1
   RUNG wire#powerrail
      { S7_Templates := "SrcType := UInt" } NE_Contact(in1 := #BR06wAlm2, in2 := 0)
   END_RUNG wire#w1
   RUNG wire#powerrail
      Contact( #BR06wAlm3.%X1 )
   END_RUNG wire#w1
   RUNG wire#powerrail
      Contact( #BR06wAlm3.%X2 )
   END_RUNG wire#w1
   RUNG wire#powerrail
      Contact( #BR06wAlm3.%X3 )
   END_RUNG wire#w1
   RUNG wire#powerrail
      Contact( #BR06wAlm3.%X4 )
   END_RUNG wire#w1
   RUNG wire#powerrail
      Contact( #BR06wAlm3.%X5 )
   END_RUNG wire#w1
   RUNG wire#powerrail
      Contact( #BR06wAlm3.%X6 )
   END_RUNG wire#w1
   RUNG wire#powerrail
      Contact( #BR06wAlm3.%X7 )
   END_RUNG wire#w1
   RUNG wire#powerrail
      Contact( #BR06wAlm3.%X10 )
   END_RUNG wire#w1
   RUNG wire#powerrail
      Contact( #BR06wAlm3.%X11 )
   END_RUNG wire#w1
   // the same network as SCL:
   "BMS1".BR06xFltSt := #BR06wAlm1.%X14 OR #BR06wAlm1.%X15 OR (#BR06wAlm2 <> 0) OR #BR06wAlm3.%X1 OR #BR06wAlm3.%X2 OR #BR06wAlm3.%X3 OR #BR06wAlm3.%X4 OR #BR06wAlm3.%X5 OR #BR06wAlm3.%X6 OR #BR06wAlm3.%X7 OR #BR06wAlm3.%X10 OR #BR06wAlm3.%X11;
END_REGION

REGION Network 93: BMS1 BR06 Alarm
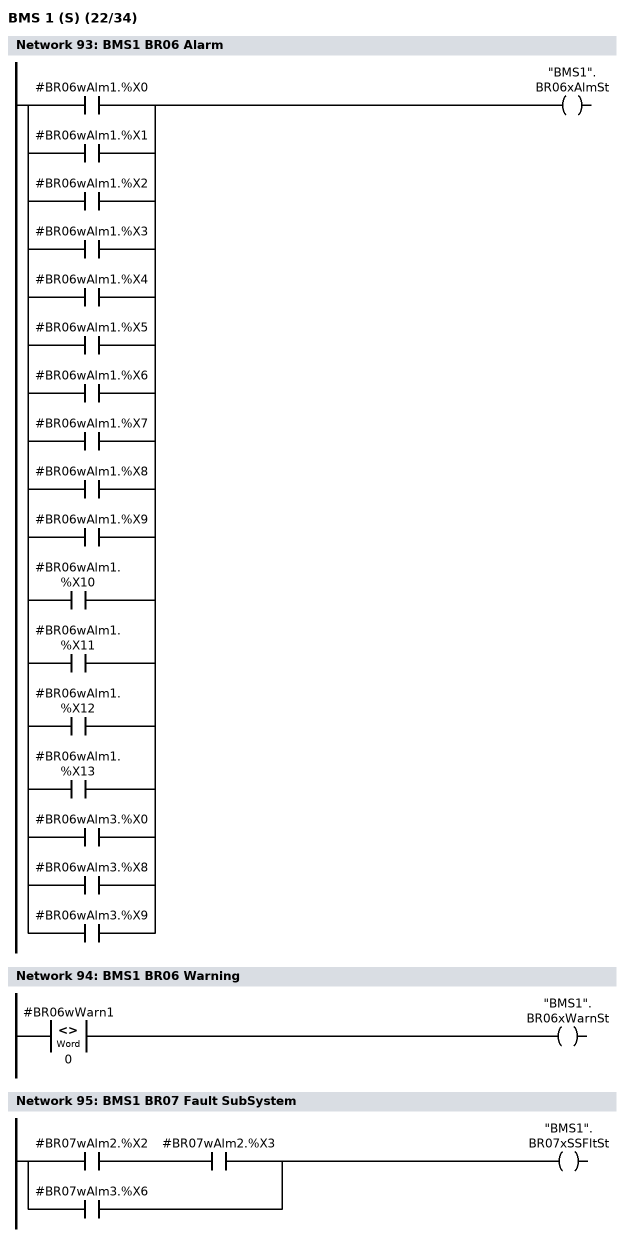
   RUNG wire#powerrail
      Contact( #BR06wAlm1.%X0 )
      wire#w1
      Coil( "BMS1".BR06xAlmSt )
   END_RUNG
   RUNG wire#powerrail
      Contact( #BR06wAlm1.%X1 )
   END_RUNG wire#w1
   RUNG wire#powerrail
      Contact( #BR06wAlm1.%X2 )
   END_RUNG wire#w1
   RUNG wire#powerrail
      Contact( #BR06wAlm1.%X3 )
   END_RUNG wire#w1
   RUNG wire#powerrail
      Contact( #BR06wAlm1.%X4 )
   END_RUNG wire#w1
   RUNG wire#powerrail
      Contact( #BR06wAlm1.%X5 )
   END_RUNG wire#w1
   RUNG wire#powerrail
      Contact( #BR06wAlm1.%X6 )
   END_RUNG wire#w1
   RUNG wire#powerrail
      Contact( #BR06wAlm1.%X7 )
   END_RUNG wire#w1
   RUNG wire#powerrail
      Contact( #BR06wAlm1.%X8 )
   END_RUNG wire#w1
   RUNG wire#powerrail
      Contact( #BR06wAlm1.%X9 )
   END_RUNG wire#w1
   RUNG wire#powerrail
      Contact( #BR06wAlm1.%X10 )
   END_RUNG wire#w1
   RUNG wire#powerrail
      Contact( #BR06wAlm1.%X11 )
   END_RUNG wire#w1
   RUNG wire#powerrail
      Contact( #BR06wAlm1.%X12 )
   END_RUNG wire#w1
   RUNG wire#powerrail
      Contact( #BR06wAlm1.%X13 )
   END_RUNG wire#w1
   RUNG wire#powerrail
      Contact( #BR06wAlm3.%X0 )
   END_RUNG wire#w1
   RUNG wire#powerrail
      Contact( #BR06wAlm3.%X8 )
   END_RUNG wire#w1
   RUNG wire#powerrail
      Contact( #BR06wAlm3.%X9 )
   END_RUNG wire#w1
   // the same network as SCL:
   "BMS1".BR06xAlmSt := #BR06wAlm1.%X0 OR #BR06wAlm1.%X1 OR #BR06wAlm1.%X2 OR #BR06wAlm1.%X3 OR #BR06wAlm1.%X4 OR #BR06wAlm1.%X5 OR #BR06wAlm1.%X6 OR #BR06wAlm1.%X7 OR #BR06wAlm1.%X8 OR #BR06wAlm1.%X9 OR #BR06wAlm1.%X10 OR #BR06wAlm1.%X11 OR #BR06wAlm1.%X12 OR #BR06wAlm1.%X13 OR #BR06wAlm3.%X0 OR #BR06wAlm3.%X8 OR #BR06wAlm3.%X9;
END_REGION

REGION Network 94: BMS1 BR06 Warning
   RUNG wire#powerrail
      { S7_Templates := "SrcType := Word" } NE_Contact(in1 := #BR06wWarn1, in2 := 0)
      Coil( "BMS1".BR06xWarnSt )
   END_RUNG
   // the same network as SCL:
   "BMS1".BR06xWarnSt := #BR06wWarn1 <> 0;
END_REGION

REGION Network 95: BMS1 BR07 Fault SubSystem
   RUNG wire#powerrail
      Contact( #BR07wAlm2.%X2 )
      Contact( #BR07wAlm2.%X3 )
      wire#w1
      Coil( "BMS1".BR07xSSFltSt )
   END_RUNG
   RUNG wire#powerrail
      Contact( #BR07wAlm3.%X6 )
   END_RUNG wire#w1
   // the same network as SCL:
   "BMS1".BR07xSSFltSt := (#BR07wAlm2.%X2 AND #BR07wAlm2.%X3) OR #BR07wAlm3.%X6;
END_REGION

REGION Network 96: BMS1 BR07 Fault
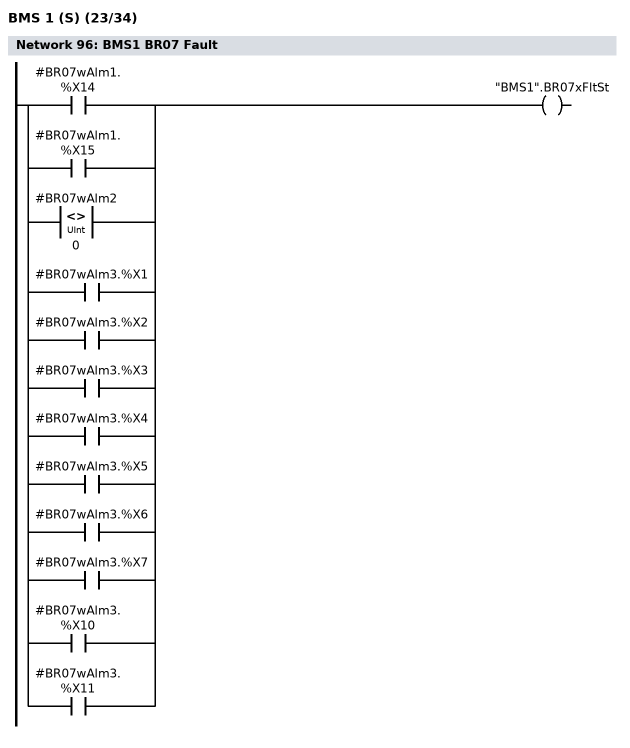
   RUNG wire#powerrail
      Contact( #BR07wAlm1.%X14 )
      wire#w1
      Coil( "BMS1".BR07xFltSt )
   END_RUNG
   RUNG wire#powerrail
      Contact( #BR07wAlm1.%X15 )
   END_RUNG wire#w1
   RUNG wire#powerrail
      { S7_Templates := "SrcType := UInt" } NE_Contact(in1 := #BR07wAlm2, in2 := 0)
   END_RUNG wire#w1
   RUNG wire#powerrail
      Contact( #BR07wAlm3.%X1 )
   END_RUNG wire#w1
   RUNG wire#powerrail
      Contact( #BR07wAlm3.%X2 )
   END_RUNG wire#w1
   RUNG wire#powerrail
      Contact( #BR07wAlm3.%X3 )
   END_RUNG wire#w1
   RUNG wire#powerrail
      Contact( #BR07wAlm3.%X4 )
   END_RUNG wire#w1
   RUNG wire#powerrail
      Contact( #BR07wAlm3.%X5 )
   END_RUNG wire#w1
   RUNG wire#powerrail
      Contact( #BR07wAlm3.%X6 )
   END_RUNG wire#w1
   RUNG wire#powerrail
      Contact( #BR07wAlm3.%X7 )
   END_RUNG wire#w1
   RUNG wire#powerrail
      Contact( #BR07wAlm3.%X10 )
   END_RUNG wire#w1
   RUNG wire#powerrail
      Contact( #BR07wAlm3.%X11 )
   END_RUNG wire#w1
   // the same network as SCL:
   "BMS1".BR07xFltSt := #BR07wAlm1.%X14 OR #BR07wAlm1.%X15 OR (#BR07wAlm2 <> 0) OR #BR07wAlm3.%X1 OR #BR07wAlm3.%X2 OR #BR07wAlm3.%X3 OR #BR07wAlm3.%X4 OR #BR07wAlm3.%X5 OR #BR07wAlm3.%X6 OR #BR07wAlm3.%X7 OR #BR07wAlm3.%X10 OR #BR07wAlm3.%X11;
END_REGION

REGION Network 97: BMS1 BR07 Alarm
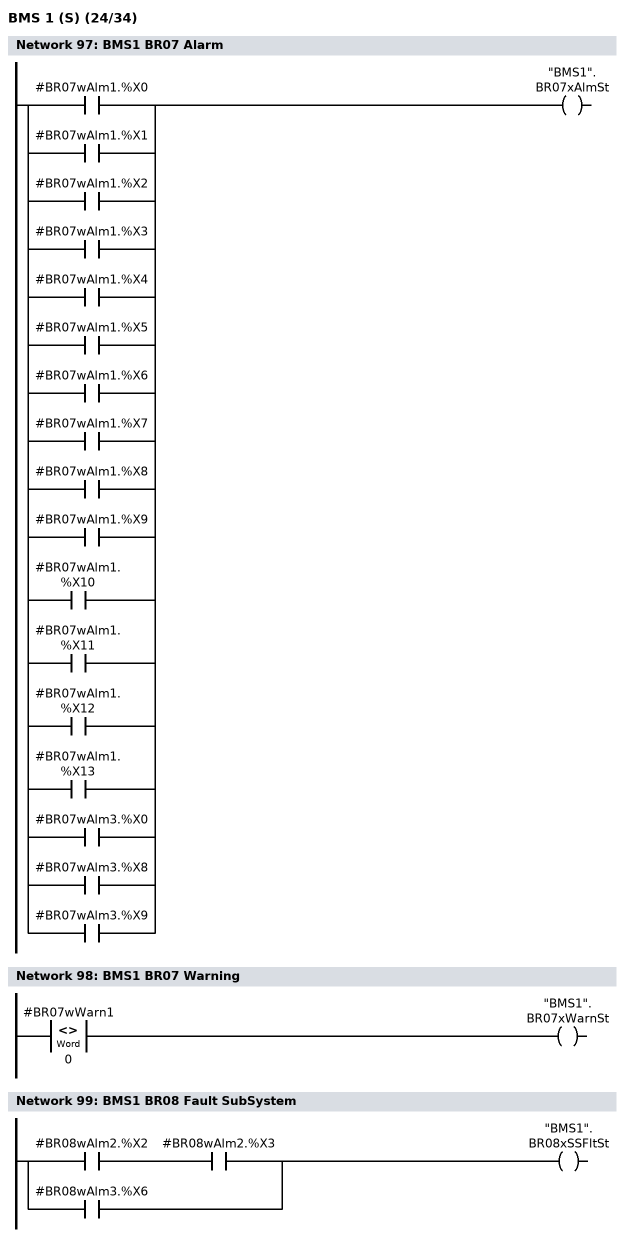
   RUNG wire#powerrail
      Contact( #BR07wAlm1.%X0 )
      wire#w1
      Coil( "BMS1".BR07xAlmSt )
   END_RUNG
   RUNG wire#powerrail
      Contact( #BR07wAlm1.%X1 )
   END_RUNG wire#w1
   RUNG wire#powerrail
      Contact( #BR07wAlm1.%X2 )
   END_RUNG wire#w1
   RUNG wire#powerrail
      Contact( #BR07wAlm1.%X3 )
   END_RUNG wire#w1
   RUNG wire#powerrail
      Contact( #BR07wAlm1.%X4 )
   END_RUNG wire#w1
   RUNG wire#powerrail
      Contact( #BR07wAlm1.%X5 )
   END_RUNG wire#w1
   RUNG wire#powerrail
      Contact( #BR07wAlm1.%X6 )
   END_RUNG wire#w1
   RUNG wire#powerrail
      Contact( #BR07wAlm1.%X7 )
   END_RUNG wire#w1
   RUNG wire#powerrail
      Contact( #BR07wAlm1.%X8 )
   END_RUNG wire#w1
   RUNG wire#powerrail
      Contact( #BR07wAlm1.%X9 )
   END_RUNG wire#w1
   RUNG wire#powerrail
      Contact( #BR07wAlm1.%X10 )
   END_RUNG wire#w1
   RUNG wire#powerrail
      Contact( #BR07wAlm1.%X11 )
   END_RUNG wire#w1
   RUNG wire#powerrail
      Contact( #BR07wAlm1.%X12 )
   END_RUNG wire#w1
   RUNG wire#powerrail
      Contact( #BR07wAlm1.%X13 )
   END_RUNG wire#w1
   RUNG wire#powerrail
      Contact( #BR07wAlm3.%X0 )
   END_RUNG wire#w1
   RUNG wire#powerrail
      Contact( #BR07wAlm3.%X8 )
   END_RUNG wire#w1
   RUNG wire#powerrail
      Contact( #BR07wAlm3.%X9 )
   END_RUNG wire#w1
   // the same network as SCL:
   "BMS1".BR07xAlmSt := #BR07wAlm1.%X0 OR #BR07wAlm1.%X1 OR #BR07wAlm1.%X2 OR #BR07wAlm1.%X3 OR #BR07wAlm1.%X4 OR #BR07wAlm1.%X5 OR #BR07wAlm1.%X6 OR #BR07wAlm1.%X7 OR #BR07wAlm1.%X8 OR #BR07wAlm1.%X9 OR #BR07wAlm1.%X10 OR #BR07wAlm1.%X11 OR #BR07wAlm1.%X12 OR #BR07wAlm1.%X13 OR #BR07wAlm3.%X0 OR #BR07wAlm3.%X8 OR #BR07wAlm3.%X9;
END_REGION

REGION Network 98: BMS1 BR07 Warning
   RUNG wire#powerrail
      { S7_Templates := "SrcType := Word" } NE_Contact(in1 := #BR07wWarn1, in2 := 0)
      Coil( "BMS1".BR07xWarnSt )
   END_RUNG
   // the same network as SCL:
   "BMS1".BR07xWarnSt := #BR07wWarn1 <> 0;
END_REGION

REGION Network 99: BMS1 BR08 Fault SubSystem
   RUNG wire#powerrail
      Contact( #BR08wAlm2.%X2 )
      Contact( #BR08wAlm2.%X3 )
      wire#w1
      Coil( "BMS1".BR08xSSFltSt )
   END_RUNG
   RUNG wire#powerrail
      Contact( #BR08wAlm3.%X6 )
   END_RUNG wire#w1
   // the same network as SCL:
   "BMS1".BR08xSSFltSt := (#BR08wAlm2.%X2 AND #BR08wAlm2.%X3) OR #BR08wAlm3.%X6;
END_REGION

REGION Network 100: BMS1 BR08 Fault
